   DATA[1296,24] := 2.0;
   DATA[1296,25] := 2.0;
   DATA[1296,26] := 7.87798;
   DATA[1296,27] := 143.0403;
   DATA[1296,28] := 263.0095;
   DATA[1296,29] := 11.88157;
   DATA[1296,30] := 1.726993;
   DATA[1296,31] := 1.274753;
   DATA[1296,32] := 0.7348846;
   DATA[1296,33] := 0.3082983;
   DATA[1296,34] := 2.0;
   DATA[1296,35] := 250.4646;
   DATA[1296,36] := 1.730048;
   DATA[1296,37] := 189.2624;
   DATA[1296,38] := 0.000128152;
   DATA[1296,39] := 1.0;
   DATA[1297,0] := 2.532428;
   DATA[1297,1] := 799.8927;
   DATA[1297,2] := 2.0;
   DATA[1297,3] := 1.0;
   DATA[1297,4] := 262.5609;
   DATA[1297,5] := 8.464369;
   DATA[1297,6] := 317.6878;
   DATA[1297,8] := 1.0;
   DATA[1297,9] := 1.0;
   DATA[1297,10] := 1.0;
   DATA[1297,11] := 1.997567;
   DATA[1297,12] := 0.000256221;
   DATA[1297,13] := 1010.879;
   DATA[1297,14] := 1.0;
   DATA[1297,15] := 1.0;
   DATA[1297,16] := 1.0;
   DATA[1297,17] := 1.0;
   DATA[1297,18] := 1.0;
   DATA[1297,19] := 1.0;
   DATA[1297,20] := 148.808;
   DATA[1297,21] := 153.8836;
   DATA[1297,22] := 1.716208;
   DATA[1297,23] := 809.6001;
   DATA[1297,24] := 2.0;
   DATA[1297,25] := 2.0;
   DATA[1297,26] := 7.87798;
   DATA[1297,27] := 143.0403;
   DATA[1297,28] := 263.0095;
   DATA[1297,29] := 12.07383;
   DATA[1297,30] := 1.726993;
   DATA[1297,31] := 1.277699;
   DATA[1297,32] := 0.7348846;
   DATA[1297,33] := 0.3082983;
   DATA[1297,34] := 2.0;
   DATA[1297,35] := 250.5447;
   DATA[1297,36] := 1.730048;
   DATA[1297,37] := 189.2624;
   DATA[1297,38] := 0.000128152;
   DATA[1297,39] := 1.0;
   DATA[1298,0] := 2.537873;
   DATA[1298,1] := 800.6385;
   DATA[1298,2] := 2.0;
   DATA[1298,3] := 1.0;
   DATA[1298,4] := 262.5609;
   DATA[1298,5] := 8.464369;
   DATA[1298,6] := 317.6878;
   DATA[1298,8] := 1.0;
   DATA[1298,9] := 1.0;
   DATA[1298,10] := 1.0;
   DATA[1298,11] := 1.997567;
   DATA[1298,12] := 0.000256221;
   DATA[1298,13] := 1010.879;
   DATA[1298,14] := 1.0;
   DATA[1298,15] := 1.0;
   DATA[1298,16] := 1.0;
   DATA[1298,17] := 1.0;
   DATA[1298,18] := 1.0;
   DATA[1298,19] := 1.0;
   DATA[1298,20] := 148.808;
   DATA[1298,21] := 153.8836;
   DATA[1298,22] := 1.716208;
   DATA[1298,23] := 809.1771;
   DATA[1298,24] := 2.0;
   DATA[1298,25] := 2.0;
   DATA[1298,26] := 7.87798;
   DATA[1298,27] := 143.0403;
   DATA[1298,28] := 263.0095;
   DATA[1298,29] := 12.07383;
   DATA[1298,30] := 1.726993;
   DATA[1298,31] := 1.274881;
   DATA[1298,32] := 0.7353967;
   DATA[1298,33] := 0.3082983;
   DATA[1298,34] := 2.0;
   DATA[1298,35] := 250.5447;
   DATA[1298,36] := 1.681991;
   DATA[1298,37] := 189.2624;
   DATA[1298,38] := 0.000128152;
   DATA[1298,39] := 1.0;
   DATA[1299,0] := 2.539474;
   DATA[1299,1] := 801.188;
   DATA[1299,3] := 1.0;
   DATA[1299,4] := 262.5609;
   DATA[1299,5] := 8.464369;
   DATA[1299,6] := 317.6878;
   DATA[1299,8] := 1.0;
   DATA[1299,9] := 1.0;
   DATA[1299,10] := 1.0;
   DATA[1299,11] := 1.997567;
   DATA[1299,12] := 0.000256221;
   DATA[1299,13] := 1010.758;
   DATA[1299,14] := 1.0;
   DATA[1299,15] := 1.0;
   DATA[1299,16] := 1.0;
   DATA[1299,17] := 1.0;
   DATA[1299,18] := 1.0;
   DATA[1299,19] := 1.0;
   DATA[1299,20] := 148.808;
   DATA[1299,21] := 153.8836;
   DATA[1299,22] := 1.717746;
   DATA[1299,23] := 809.1387;
   DATA[1299,24] := 2.0;
   DATA[1299,25] := 2.0;
   DATA[1299,26] := 7.87798;
   DATA[1299,27] := 143.0403;
   DATA[1299,28] := 263.0095;
   DATA[1299,29] := 12.07383;
   DATA[1299,30] := 1.726993;
   DATA[1299,31] := 1.291149;
   DATA[1299,32] := 0.7353967;
   DATA[1299,33] := 0.3082983;
   DATA[1299,34] := 2.0;
   DATA[1299,35] := 250.3525;
   DATA[1299,36] := 1.681991;
   DATA[1299,37] := 189.2624;
   DATA[1299,38] := 0.000128152;
   DATA[1299,39] := 1.0;
   DATA[1300,0] := 2.544278;
   DATA[1300,1] := 801.8161;
   DATA[1300,3] := 1.0;
   DATA[1300,4] := 262.5609;
   DATA[1300,5] := 8.464369;
   DATA[1300,6] := 317.6878;
   DATA[1300,8] := 1.0;
   DATA[1300,9] := 1.0;
   DATA[1300,10] := 1.0;
   DATA[1300,11] := 2.010372;
   DATA[1300,12] := 0.000256221;
   DATA[1300,13] := 1010.558;
   DATA[1300,14] := 1.0;
   DATA[1300,15] := 1.0;
   DATA[1300,16] := 1.0;
   DATA[1300,17] := 1.0;
   DATA[1300,18] := 1.0;
   DATA[1300,19] := 1.0;
   DATA[1300,20] := 148.808;
   DATA[1300,21] := 153.6785;
   DATA[1300,22] := 1.717746;
   DATA[1300,23] := 808.5619;
   DATA[1300,24] := 2.0;
   DATA[1300,25] := 2.0;
   DATA[1300,26] := 7.87798;
   DATA[1300,27] := 143.0403;
   DATA[1300,28] := 263.0095;
   DATA[1300,29] := 12.07383;
   DATA[1300,30] := 1.726993;
   DATA[1300,31] := 1.289996;
   DATA[1300,32] := 0.7353967;
   DATA[1300,33] := 0.3082983;
   DATA[1300,34] := 2.0;
   DATA[1300,35] := 250.3525;
   DATA[1300,36] := 1.681991;
   DATA[1300,37] := 189.2624;
   DATA[1300,38] := 0.000128152;
   DATA[1300,39] := 1.0;
   DATA[1301,0] := 2.54652;
   DATA[1301,1] := 802.5619;
   DATA[1301,3] := 1.0;
   DATA[1301,4] := 262.5609;
   DATA[1301,5] := 8.464369;
   DATA[1301,6] := 317.6878;
   DATA[1301,8] := 1.0;
   DATA[1301,9] := 1.0;
   DATA[1301,10] := 1.0;
   DATA[1301,11] := 2.010372;
   DATA[1301,12] := 0.000256221;
   DATA[1301,13] := 1010.678;
   DATA[1301,14] := 1.0;
   DATA[1301,15] := 1.0;
   DATA[1301,16] := 1.0;
   DATA[1301,17] := 1.0;
   DATA[1301,18] := 1.0;
   DATA[1301,19] := 1.0;
   DATA[1301,20] := 148.808;
   DATA[1301,21] := 153.6785;
   DATA[1301,22] := 1.717746;
   DATA[1301,23] := 808.1774;
   DATA[1301,24] := 2.0;
   DATA[1301,25] := 2.0;
   DATA[1301,26] := 7.87798;
   DATA[1301,27] := 143.0403;
   DATA[1301,28] := 263.0095;
   DATA[1301,29] := 12.07383;
   DATA[1301,30] := 1.726352;
   DATA[1301,31] := 1.28167;
   DATA[1301,32] := 0.7353967;
   DATA[1301,33] := 0.3082983;
   DATA[1301,34] := 2.0;
   DATA[1301,35] := 250.3525;
   DATA[1301,36] := 1.681991;
   DATA[1301,37] := 189.2624;
   DATA[1301,38] := 0.000128152;
   DATA[1301,39] := 1.0;
   DATA[1302,0] := 2.548762;
   DATA[1302,1] := 802.9544;
   DATA[1302,3] := 1.0;
   DATA[1302,4] := 262.5609;
   DATA[1302,5] := 8.464369;
   DATA[1302,6] := 317.6878;
   DATA[1302,8] := 1.0;
   DATA[1302,9] := 1.0;
   DATA[1302,10] := 1.0;
   DATA[1302,11] := 2.010372;
   DATA[1302,12] := 0.000256221;
   DATA[1302,13] := 1010.558;
   DATA[1302,14] := 1.0;
   DATA[1302,15] := 1.0;
   DATA[1302,16] := 1.0;
   DATA[1302,17] := 1.0;
   DATA[1302,18] := 1.0;
   DATA[1302,19] := 1.0;
   DATA[1302,20] := 148.808;
   DATA[1302,21] := 153.6785;
   DATA[1302,22] := 1.717746;
   DATA[1302,23] := 807.8313;
   DATA[1302,24] := 2.0;
   DATA[1302,25] := 2.0;
   DATA[1302,26] := 7.87798;
   DATA[1302,27] := 143.0403;
   DATA[1302,28] := 263.0095;
   DATA[1302,29] := 12.07383;
   DATA[1302,30] := 1.724686;
   DATA[1302,31] := 1.28167;
   DATA[1302,32] := 0.7353967;
   DATA[1302,33] := 0.3082983;
   DATA[1302,34] := 2.0;
   DATA[1302,35] := 250.3525;
   DATA[1302,36] := 1.681991;
   DATA[1302,37] := 189.2624;
   DATA[1302,38] := 0.000128152;
   DATA[1302,39] := 1.0;
   DATA[1303,0] := 2.548762;
   DATA[1303,1] := 803.9357;
   DATA[1303,3] := 1.0;
   DATA[1303,4] := 262.5609;
   DATA[1303,5] := 8.464369;
   DATA[1303,6] := 317.6878;
   DATA[1303,8] := 1.0;
   DATA[1303,9] := 1.0;
   DATA[1303,10] := 1.0;
   DATA[1303,11] := 2.010372;
   DATA[1303,12] := 0.000256221;
   DATA[1303,13] := 1010.678;
   DATA[1303,14] := 1.0;
   DATA[1303,15] := 1.0;
   DATA[1303,16] := 1.0;
   DATA[1303,17] := 1.0;
   DATA[1303,18] := 1.0;
   DATA[1303,19] := 1.0;
   DATA[1303,20] := 148.808;
   DATA[1303,21] := 153.6785;
   DATA[1303,22] := 1.717746;
   DATA[1303,23] := 807.4468;
   DATA[1303,24] := 2.0;
   DATA[1303,25] := 2.0;
   DATA[1303,26] := 7.87798;
   DATA[1303,27] := 143.0403;
   DATA[1303,28] := 263.0095;
   DATA[1303,29] := 12.07383;
   DATA[1303,30] := 1.724686;
   DATA[1303,31] := 1.274497;
   DATA[1303,32] := 0.7353967;
   DATA[1303,33] := 0.3082983;
   DATA[1303,34] := 2.0;
   DATA[1303,35] := 250.3525;
   DATA[1303,36] := 1.681991;
   DATA[1303,37] := 189.2624;
   DATA[1303,38] := 0.000128152;
   DATA[1303,39] := 1.0;
   DATA[1304,0] := 2.537873;
   DATA[1304,1] := 804.4068;
   DATA[1304,3] := 1.0;
   DATA[1304,4] := 262.5609;
   DATA[1304,5] := 8.464369;
   DATA[1304,6] := 317.6878;
   DATA[1304,8] := 1.0;
   DATA[1304,9] := 1.0;
   DATA[1304,10] := 1.0;
   DATA[1304,11] := 2.010372;
   DATA[1304,12] := 0.000256221;
   DATA[1304,13] := 1010.959;
   DATA[1304,14] := 1.0;
   DATA[1304,15] := 1.0;
   DATA[1304,16] := 1.0;
   DATA[1304,17] := 1.0;
   DATA[1304,18] := 1.0;
   DATA[1304,19] := 1.0;
   DATA[1304,20] := 148.808;
   DATA[1304,21] := 153.6785;
   DATA[1304,22] := 1.717746;
   DATA[1304,23] := 807.4853;
   DATA[1304,24] := 2.0;
   DATA[1304,25] := 2.0;
   DATA[1304,26] := 7.87798;
   DATA[1304,27] := 143.0403;
   DATA[1304,28] := 263.0095;
   DATA[1304,29] := 12.07383;
   DATA[1304,30] := 1.724686;
   DATA[1304,31] := 1.277315;
   DATA[1304,32] := 0.7353967;
   DATA[1304,33] := 0.3082983;
   DATA[1304,34] := 2.0;
   DATA[1304,35] := 250.3525;
   DATA[1304,36] := 1.681991;
   DATA[1304,37] := 189.2624;
   DATA[1304,38] := 0.000128152;
   DATA[1304,39] := 1.0;
   DATA[1305,0] := 2.515133;
   DATA[1305,1] := 804.9171;
   DATA[1305,3] := 1.0;
   DATA[1305,4] := 262.5609;
   DATA[1305,5] := 8.464369;
   DATA[1305,6] := 317.6878;
   DATA[1305,8] := 1.0;
   DATA[1305,9] := 1.0;
   DATA[1305,10] := 1.0;
   DATA[1305,11] := 2.010372;
   DATA[1305,12] := 0.000256221;
   DATA[1305,13] := 1010.919;
   DATA[1305,14] := 1.0;
   DATA[1305,15] := 1.0;
   DATA[1305,16] := 1.0;
   DATA[1305,17] := 1.0;
   DATA[1305,18] := 1.0;
   DATA[1305,19] := 1.0;
   DATA[1305,20] := 148.808;
   DATA[1305,21] := 153.6785;
   DATA[1305,22] := 1.717746;
   DATA[1305,23] := 806.9085;
   DATA[1305,24] := 2.0;
   DATA[1305,25] := 2.0;
   DATA[1305,26] := 7.87798;
   DATA[1305,27] := 143.0403;
   DATA[1305,28] := 263.0095;
   DATA[1305,29] := 12.07383;
   DATA[1305,30] := 1.724686;
   DATA[1305,31] := 1.291789;
   DATA[1305,32] := 0.7353967;
   DATA[1305,33] := 0.3082983;
   DATA[1305,34] := 2.0;
   DATA[1305,35] := 250.3525;
   DATA[1305,36] := 1.681991;
   DATA[1305,37] := 189.2624;
   DATA[1305,38] := 0.000128152;
   DATA[1305,39] := 1.0;
   DATA[1306,0] := 2.464209;
   DATA[1306,1] := 805.5451;
   DATA[1306,3] := 1.0;
   DATA[1306,4] := 262.5609;
   DATA[1306,5] := 8.464369;
   DATA[1306,6] := 317.6878;
   DATA[1306,8] := 1.0;
   DATA[1306,9] := 1.0;
   DATA[1306,10] := 1.0;
   DATA[1306,11] := 2.010372;
   DATA[1306,12] := 0.000256221;
   DATA[1306,13] := 1011.119;
   DATA[1306,14] := 1.0;
   DATA[1306,15] := 1.0;
   DATA[1306,16] := 1.0;
   DATA[1306,17] := 1.0;
   DATA[1306,18] := 1.0;
   DATA[1306,19] := 1.0;
   DATA[1306,20] := 148.808;
   DATA[1306,21] := 153.6785;
   DATA[1306,22] := 1.717746;
   DATA[1306,23] := 806.2933;
   DATA[1306,24] := 2.0;
   DATA[1306,25] := 2.0;
   DATA[1306,26] := 7.87798;
   DATA[1306,27] := 143.0403;
   DATA[1306,28] := 263.0095;
   DATA[1306,29] := 12.07383;
   DATA[1306,30] := 1.724686;
   DATA[1306,31] := 1.301652;
   DATA[1306,32] := 0.7353967;
   DATA[1306,33] := 0.3082983;
   DATA[1306,34] := 2.0;
   DATA[1306,35] := 250.3525;
   DATA[1306,36] := 1.746067;
   DATA[1306,37] := 189.2624;
   DATA[1306,38] := 0.000128152;
   DATA[1306,39] := 1.0;
   DATA[1307,0] := 2.393428;
   DATA[1307,1] := 805.9769;
   DATA[1307,2] := 1.0;
   DATA[1307,3] := 1.0;
   DATA[1307,4] := 262.5609;
   DATA[1307,5] := 8.464369;
   DATA[1307,6] := 317.6878;
   DATA[1307,8] := 1.0;
   DATA[1307,9] := 1.0;
   DATA[1307,10] := 1.0;
   DATA[1307,11] := 2.010372;
   DATA[1307,12] := 0.000256221;
   DATA[1307,13] := 1010.758;
   DATA[1307,14] := 1.0;
   DATA[1307,15] := 1.0;
   DATA[1307,16] := 1.0;
   DATA[1307,17] := 1.0;
   DATA[1307,18] := 1.0;
   DATA[1307,19] := 1.0;
   DATA[1307,20] := 148.808;
   DATA[1307,21] := 153.8067;
   DATA[1307,22] := 1.717746;
   DATA[1307,23] := 805.7934;
   DATA[1307,24] := 2.0;
   DATA[1307,25] := 2.0;
   DATA[1307,26] := 7.87798;
   DATA[1307,27] := 143.0403;
   DATA[1307,28] := 263.0095;
   DATA[1307,29] := 12.07383;
   DATA[1307,30] := 1.724686;
   DATA[1307,31] := 1.302677;
   DATA[1307,32] := 0.7353967;
   DATA[1307,33] := 0.3082983;
   DATA[1307,34] := 2.0;
   DATA[1307,35] := 250.3525;
   DATA[1307,36] := 1.746067;
   DATA[1307,37] := 189.2624;
   DATA[1307,38] := 0.000128152;
   DATA[1307,39] := 1.0;
   DATA[1308,0] := 2.276206;
   DATA[1308,1] := 806.2516;
   DATA[1308,2] := 1.0;
   DATA[1308,3] := 1.0;
   DATA[1308,4] := 262.5609;
   DATA[1308,5] := 8.464369;
   DATA[1308,6] := 317.6878;
   DATA[1308,8] := 1.0;
   DATA[1308,9] := 1.0;
   DATA[1308,10] := 1.0;
   DATA[1308,11] := 2.010372;
   DATA[1308,12] := 0.000256221;
   DATA[1308,13] := 1011.079;
   DATA[1308,14] := 1.0;
   DATA[1308,15] := 1.0;
   DATA[1308,16] := 1.0;
   DATA[1308,17] := 1.0;
   DATA[1308,18] := 1.0;
   DATA[1308,19] := 1.0;
   DATA[1308,20] := 148.808;
   DATA[1308,21] := 153.8067;
   DATA[1308,22] := 1.717746;
   DATA[1308,23] := 805.7934;
   DATA[1308,24] := 2.0;
   DATA[1308,25] := 2.0;
   DATA[1308,26] := 7.87798;
   DATA[1308,27] := 143.0403;
   DATA[1308,28] := 263.0095;
   DATA[1308,29] := 12.07383;
   DATA[1308,30] := 1.724686;
   DATA[1308,31] := 1.310747;
   DATA[1308,32] := 0.7353967;
   DATA[1308,33] := 0.3082983;
   DATA[1308,34] := 2.0;
   DATA[1308,35] := 250.3525;
   DATA[1308,36] := 1.746067;
   DATA[1308,37] := 189.2624;
   DATA[1308,38] := 0.000128152;
   DATA[1308,39] := 1.0;
   DATA[1309,0] := 2.053935;
   DATA[1309,1] := 806.6442;
   DATA[1309,2] := 1.0;
   DATA[1309,3] := 1.0;
   DATA[1309,4] := 262.5609;
   DATA[1309,5] := 8.464369;
   DATA[1309,6] := 317.6878;
   DATA[1309,8] := 1.0;
   DATA[1309,9] := 1.0;
   DATA[1309,10] := 1.0;
   DATA[1309,11] := 2.010372;
   DATA[1309,12] := 0.000256221;
   DATA[1309,13] := 1011.159;
   DATA[1309,14] := 1.0;
   DATA[1309,15] := 1.0;
   DATA[1309,16] := 1.0;
   DATA[1309,17] := 1.0;
   DATA[1309,18] := 1.0;
   DATA[1309,19] := 1.0;
   DATA[1309,20] := 148.808;
   DATA[1309,21] := 153.8067;
   DATA[1309,22] := 1.717746;
   DATA[1309,23] := 805.1397;
   DATA[1309,24] := 2.0;
   DATA[1309,25] := 2.0;
   DATA[1309,26] := 7.87798;
   DATA[1309,27] := 143.0403;
   DATA[1309,28] := 263.0095;
   DATA[1309,29] := 12.07383;
   DATA[1309,30] := 1.724045;
   DATA[1309,31] := 1.312028;
   DATA[1309,32] := 0.7353967;
   DATA[1309,33] := 0.3082983;
   DATA[1309,34] := 2.0;
   DATA[1309,35] := 250.3525;
   DATA[1309,36] := 1.746067;
   DATA[1309,37] := 189.2624;
   DATA[1309,38] := 0.000128152;
   DATA[1309,39] := 1.0;
   DATA[1310,0] := 1.653268;
   DATA[1310,1] := 807.3115;
   DATA[1310,2] := 1.0;
   DATA[1310,3] := 1.0;
   DATA[1310,4] := 262.5609;
   DATA[1310,5] := 8.464369;
   DATA[1310,6] := 317.6878;
   DATA[1310,8] := 1.0;
   DATA[1310,9] := 1.0;
   DATA[1310,10] := 1.0;
   DATA[1310,11] := 2.010372;
   DATA[1310,12] := 0.000256221;
   DATA[1310,13] := 1010.678;
   DATA[1310,14] := 1.0;
   DATA[1310,15] := 1.0;
   DATA[1310,16] := 1.0;
   DATA[1310,17] := 1.0;
   DATA[1310,18] := 1.0;
   DATA[1310,19] := 1.0;
   DATA[1310,20] := 148.808;
   DATA[1310,21] := 153.8067;
   DATA[1310,22] := 1.717746;
   DATA[1310,23] := 804.6398;
   DATA[1310,24] := 2.0;
   DATA[1310,25] := 2.0;
   DATA[1310,26] := 7.87798;
   DATA[1310,27] := 143.0403;
   DATA[1310,28] := 263.0095;
   DATA[1310,29] := 12.07383;
   DATA[1310,30] := 1.724045;
   DATA[1310,31] := 1.305367;
   DATA[1310,32] := 0.7353967;
   DATA[1310,33] := 0.3082983;
   DATA[1310,34] := 2.0;
   DATA[1310,35] := 250.3525;
   DATA[1310,36] := 1.746067;
   DATA[1310,37] := 189.2624;
   DATA[1310,38] := 0.000128152;
   DATA[1310,39] := 1.0;
   DATA[1311,0] := 1.308651;
   DATA[1311,1] := 807.7432;
   DATA[1311,2] := 1.0;
   DATA[1311,3] := 1.0;
   DATA[1311,4] := 262.5609;
   DATA[1311,5] := 8.464369;
   DATA[1311,6] := 317.6878;
   DATA[1311,8] := 1.0;
   DATA[1311,9] := 1.0;
   DATA[1311,10] := 1.0;
   DATA[1311,11] := 2.010372;
   DATA[1311,12] := 0.000256221;
   DATA[1311,13] := 1010.879;
   DATA[1311,14] := 1.0;
   DATA[1311,15] := 1.0;
   DATA[1311,16] := 1.0;
   DATA[1311,17] := 1.0;
   DATA[1311,18] := 1.0;
   DATA[1311,19] := 1.0;
   DATA[1311,20] := 148.808;
   DATA[1311,21] := 153.8067;
   DATA[1311,22] := 1.717746;
   DATA[1311,23] := 804.0246;
   DATA[1311,24] := 2.0;
   DATA[1311,25] := 2.0;
   DATA[1311,26] := 7.87798;
   DATA[1311,27] := 143.0403;
   DATA[1311,28] := 263.0095;
   DATA[1311,29] := 12.07383;
   DATA[1311,30] := 1.724045;
   DATA[1311,31] := 1.302805;
   DATA[1311,32] := 0.7353967;
   DATA[1311,33] := 0.3084265;
   DATA[1311,34] := 2.0;
   DATA[1311,35] := 250.3525;
   DATA[1311,36] := 1.746067;
   DATA[1311,37] := 189.2624;
   DATA[1311,38] := 0.000128152;
   DATA[1311,39] := 1.0;
   DATA[1312,0] := 0.9060628;
   DATA[1312,1] := 808.2928;
   DATA[1312,2] := 1.0;
   DATA[1312,3] := 1.0;
   DATA[1312,4] := 262.5609;
   DATA[1312,5] := 8.464369;
   DATA[1312,6] := 317.6878;
   DATA[1312,8] := 1.0;
   DATA[1312,9] := 1.0;
   DATA[1312,10] := 1.0;
   DATA[1312,11] := 2.010372;
   DATA[1312,13] := 1010.638;
   DATA[1312,14] := 1.0;
   DATA[1312,15] := 1.0;
   DATA[1312,16] := 1.0;
   DATA[1312,17] := 1.0;
   DATA[1312,18] := 1.0;
   DATA[1312,19] := 1.0;
   DATA[1312,20] := 148.808;
   DATA[1312,21] := 153.8067;
   DATA[1312,22] := 1.717489;
   DATA[1312,23] := 804.0246;
   DATA[1312,24] := 2.0;
   DATA[1312,25] := 2.0;
   DATA[1312,26] := 7.87798;
   DATA[1312,27] := 143.0403;
   DATA[1312,28] := 263.0095;
   DATA[1312,29] := 12.07383;
   DATA[1312,30] := 1.722123;
   DATA[1312,31] := 1.282567;
   DATA[1312,32] := 0.7353967;
   DATA[1312,33] := 0.3084265;
   DATA[1312,34] := 2.0;
   DATA[1312,35] := 250.3525;
   DATA[1312,36] := 1.746067;
   DATA[1312,37] := 189.1662;
   DATA[1312,38] := 0.000128152;
   DATA[1312,39] := 1.0;
   DATA[1313,0] := 0.5736156;
   DATA[1313,1] := 808.7245;
   DATA[1313,2] := 1.0;
   DATA[1313,3] := 1.0;
   DATA[1313,4] := 262.5609;
   DATA[1313,5] := 8.464369;
   DATA[1313,6] := 317.6878;
   DATA[1313,8] := 1.0;
   DATA[1313,9] := 1.0;
   DATA[1313,10] := 1.0;
   DATA[1313,11] := 2.010372;
   DATA[1313,13] := 1011.079;
   DATA[1313,14] := 1.0;
   DATA[1313,15] := 1.0;
   DATA[1313,16] := 1.0;
   DATA[1313,17] := 1.0;
   DATA[1313,18] := 1.0;
   DATA[1313,19] := 1.0;
   DATA[1313,20] := 148.808;
   DATA[1313,21] := 153.8067;
   DATA[1313,22] := 1.715439;
   DATA[1313,23] := 803.1786;
   DATA[1313,24] := 2.0;
   DATA[1313,25] := 2.0;
   DATA[1313,26] := 7.87798;
   DATA[1313,27] := 143.0403;
   DATA[1313,28] := 263.0095;
   DATA[1313,29] := 12.07383;
   DATA[1313,30] := 1.722123;
   DATA[1313,31] := 1.261688;
   DATA[1313,32] := 0.7353967;
   DATA[1313,33] := 0.3084265;
   DATA[1313,34] := 2.0;
   DATA[1313,35] := 250.0961;
   DATA[1313,36] := 1.746067;
   DATA[1313,37] := 188.9259;
   DATA[1313,38] := 0.000128152;
   DATA[1313,39] := 1.0;
   DATA[1314,0] := 0.3468597;
   DATA[1314,1] := 809.5096;
   DATA[1314,2] := 1.0;
   DATA[1314,3] := 1.0;
   DATA[1314,4] := 262.5609;
   DATA[1314,5] := 8.464369;
   DATA[1314,6] := 317.7903;
   DATA[1314,8] := 1.0;
   DATA[1314,9] := 1.0;
   DATA[1314,10] := 1.0;
   DATA[1314,11] := 2.010372;
   DATA[1314,13] := 1010.839;
   DATA[1314,14] := 1.0;
   DATA[1314,15] := 1.0;
   DATA[1314,16] := 1.0;
   DATA[1314,17] := 1.0;
   DATA[1314,18] := 1.0;
   DATA[1314,19] := 1.0;
   DATA[1314,20] := 148.808;
   DATA[1314,21] := 153.8067;
   DATA[1314,22] := 1.711979;
   DATA[1314,23] := 803.0248;
   DATA[1314,24] := 2.0;
   DATA[1314,25] := 2.0;
   DATA[1314,26] := 7.87798;
   DATA[1314,27] := 143.0403;
   DATA[1314,28] := 263.0095;
   DATA[1314,29] := 12.07383;
   DATA[1314,30] := 1.722123;
   DATA[1314,31] := 1.254643;
   DATA[1314,32] := 0.7353967;
   DATA[1314,33] := 0.3084265;
   DATA[1314,34] := 2.0;
   DATA[1314,35] := 249.9359;
   DATA[1314,36] := 1.778105;
   DATA[1314,37] := 188.8138;
   DATA[1314,38] := 0.000128152;
   DATA[1314,39] := 1.0;
   DATA[1315,0] := 0.1896038;
   DATA[1315,1] := 810.2162;
   DATA[1315,2] := 1.0;
   DATA[1315,3] := 1.0;
   DATA[1315,4] := 262.5609;
   DATA[1315,5] := 8.464369;
   DATA[1315,6] := 317.7903;
   DATA[1315,8] := 1.0;
   DATA[1315,9] := 1.0;
   DATA[1315,10] := 1.0;
   DATA[1315,11] := 2.010372;
   DATA[1315,13] := 1011.119;
   DATA[1315,14] := 1.0;
   DATA[1315,15] := 1.0;
   DATA[1315,16] := 1.0;
   DATA[1315,17] := 1.0;
   DATA[1315,18] := 1.0;
   DATA[1315,19] := 1.0;
   DATA[1315,20] := 148.808;
   DATA[1315,21] := 153.8067;
   DATA[1315,22] := 1.711338;
   DATA[1315,23] := 802.6788;
   DATA[1315,24] := 2.0;
   DATA[1315,25] := 2.0;
   DATA[1315,26] := 7.87798;
   DATA[1315,27] := 143.0403;
   DATA[1315,28] := 263.0095;
   DATA[1315,29] := 12.07383;
   DATA[1315,30] := 1.722123;
   DATA[1315,31] := 1.261048;
   DATA[1315,32] := 0.7353967;
   DATA[1315,33] := 0.3084265;
   DATA[1315,34] := 2.0;
   DATA[1315,35] := 249.9359;
   DATA[1315,36] := 1.778105;
   DATA[1315,37] := 188.8138;
   DATA[1315,38] := 0.000128152;
   DATA[1315,39] := 1.0;
   DATA[1316,0] := 0.09191941;
   DATA[1316,1] := 810.6087;
   DATA[1316,2] := 1.0;
   DATA[1316,3] := 1.0;
   DATA[1316,4] := 262.5609;
   DATA[1316,5] := 8.464369;
   DATA[1316,6] := 317.7903;
   DATA[1316,8] := 1.0;
   DATA[1316,9] := 1.0;
   DATA[1316,10] := 1.0;
   DATA[1316,11] := 2.010372;
   DATA[1316,13] := 1010.839;
   DATA[1316,14] := 1.0;
   DATA[1316,15] := 1.0;
   DATA[1316,16] := 1.0;
   DATA[1316,17] := 1.0;
   DATA[1316,18] := 1.0;
   DATA[1316,19] := 1.0;
   DATA[1316,20] := 148.808;
   DATA[1316,21] := 153.8067;
   DATA[1316,22] := 1.710698;
   DATA[1316,23] := 801.9098;
   DATA[1316,24] := 2.0;
   DATA[1316,25] := 2.0;
   DATA[1316,26] := 7.87798;
   DATA[1316,27] := 143.0403;
   DATA[1316,28] := 263.0095;
   DATA[1316,29] := 12.07383;
   DATA[1316,30] := 1.722123;
   DATA[1316,31] := 1.270655;
   DATA[1316,32] := 0.7353967;
   DATA[1316,33] := 0.3104122;
   DATA[1316,34] := 2.0;
   DATA[1316,35] := 249.9359;
   DATA[1316,36] := 1.778105;
   DATA[1316,37] := 188.8138;
   DATA[1316,38] := 0.000128152;
   DATA[1316,39] := 1.0;
   DATA[1317,0] := 0.0425968;
   DATA[1317,1] := 810.805;
   DATA[1317,2] := 1.0;
   DATA[1317,3] := 1.0;
   DATA[1317,4] := 262.5609;
   DATA[1317,5] := 8.464369;
   DATA[1317,6] := 317.7903;
   DATA[1317,8] := 1.0;
   DATA[1317,9] := 1.0;
   DATA[1317,10] := 1.0;
   DATA[1317,11] := 2.010372;
   DATA[1317,13] := 1010.678;
   DATA[1317,14] := 1.0;
   DATA[1317,15] := 1.0;
   DATA[1317,16] := 1.0;
   DATA[1317,17] := 1.0;
   DATA[1317,18] := 1.0;
   DATA[1317,19] := 1.0;
   DATA[1317,20] := 148.808;
   DATA[1317,21] := 153.8067;
   DATA[1317,22] := 1.710698;
   DATA[1317,23] := 801.1407;
   DATA[1317,24] := 2.0;
   DATA[1317,25] := 2.0;
   DATA[1317,26] := 7.87798;
   DATA[1317,27] := 143.0403;
   DATA[1317,28] := 263.0095;
   DATA[1317,29] := 12.07383;
   DATA[1317,30] := 1.722123;
   DATA[1317,31] := 1.27232;
   DATA[1317,32] := 0.7353967;
   DATA[1317,33] := 0.3106684;
   DATA[1317,34] := 2.0;
   DATA[1317,35] := 249.9359;
   DATA[1317,36] := 1.778105;
   DATA[1317,37] := 188.8138;
   DATA[1317,38] := 0.000128152;
   DATA[1317,39] := 1.0;
   DATA[1318,0] := 0.001281107;
   DATA[1318,1] := 811.0797;
   DATA[1318,2] := 1.0;
   DATA[1318,3] := 1.0;
   DATA[1318,4] := 262.5609;
   DATA[1318,5] := 8.464369;
   DATA[1318,6] := 317.7903;
   DATA[1318,8] := 1.0;
   DATA[1318,9] := 1.0;
   DATA[1318,10] := 1.0;
   DATA[1318,11] := 2.010372;
   DATA[1318,13] := 1011.039;
   DATA[1318,14] := 1.0;
   DATA[1318,15] := 1.0;
   DATA[1318,16] := 1.0;
   DATA[1318,17] := 1.0;
   DATA[1318,18] := 1.0;
   DATA[1318,19] := 1.0;
   DATA[1318,20] := 148.808;
   DATA[1318,21] := 153.8067;
   DATA[1318,22] := 1.710698;
   DATA[1318,23] := 800.8716;
   DATA[1318,24] := 2.0;
   DATA[1318,25] := 2.0;
   DATA[1318,26] := 7.87798;
   DATA[1318,27] := 143.0403;
   DATA[1318,28] := 263.0095;
   DATA[1318,29] := 12.07383;
   DATA[1318,30] := 1.722123;
   DATA[1318,31] := 1.27232;
   DATA[1318,32] := 0.7353967;
   DATA[1318,33] := 0.3106684;
   DATA[1318,34] := 2.0;
   DATA[1318,35] := 249.8718;
   DATA[1318,36] := 1.778105;
   DATA[1318,37] := 188.8138;
   DATA[1318,38] := 0.000128152;
   DATA[1318,39] := 1.0;
   DATA[1319,0] := 0.000640553;
   DATA[1319,1] := 811.6685;
   DATA[1319,2] := 1.0;
   DATA[1319,3] := 1.0;
   DATA[1319,4] := 262.5609;
   DATA[1319,5] := 8.464369;
   DATA[1319,6] := 317.7903;
   DATA[1319,8] := 1.0;
   DATA[1319,9] := 1.0;
   DATA[1319,10] := 1.0;
   DATA[1319,11] := 2.010372;
   DATA[1319,12] := 0.000384332;
   DATA[1319,13] := 1010.919;
   DATA[1319,14] := 1.0;
   DATA[1319,15] := 1.0;
   DATA[1319,16] := 1.0;
   DATA[1319,17] := 1.0;
   DATA[1319,18] := 1.0;
   DATA[1319,19] := 1.0;
   DATA[1319,20] := 148.808;
   DATA[1319,21] := 153.8067;
   DATA[1319,22] := 1.710698;
   DATA[1319,23] := 800.1794;
   DATA[1319,24] := 2.0;
   DATA[1319,25] := 2.0;
   DATA[1319,26] := 7.87798;
   DATA[1319,27] := 143.1684;
   DATA[1319,28] := 263.0095;
   DATA[1319,29] := 12.07383;
   DATA[1319,30] := 1.722123;
   DATA[1319,31] := 1.27232;
   DATA[1319,32] := 0.7353967;
   DATA[1319,33] := 0.3106684;
   DATA[1319,34] := 2.0;
   DATA[1319,35] := 249.8718;
   DATA[1319,36] := 1.617916;
   DATA[1319,37] := 188.6055;
   DATA[1319,38] := 0.000128152;
   DATA[1319,39] := 1.0;
   DATA[1320,1] := 812.2181;
   DATA[1320,2] := 1.0;
   DATA[1320,3] := 1.0;
   DATA[1320,4] := 262.5609;
   DATA[1320,5] := 8.464369;
   DATA[1320,6] := 318.0723;
   DATA[1320,8] := 1.0;
   DATA[1320,9] := 1.0;
   DATA[1320,10] := 1.0;
   DATA[1320,11] := 2.010372;
   DATA[1320,12] := 0.000384332;
   DATA[1320,13] := 1011.159;
   DATA[1320,14] := 1.0;
   DATA[1320,15] := 1.0;
   DATA[1320,16] := 1.0;
   DATA[1320,17] := 1.0;
   DATA[1320,18] := 1.0;
   DATA[1320,19] := 1.0;
   DATA[1320,20] := 148.808;
   DATA[1320,21] := 154.0118;
   DATA[1320,22] := 1.710698;
   DATA[1320,23] := 799.9872;
   DATA[1320,24] := 2.0;
   DATA[1320,25] := 2.0;
   DATA[1320,26] := 7.87798;
   DATA[1320,27] := 143.1684;
   DATA[1320,28] := 263.0095;
   DATA[1320,29] := 12.07383;
   DATA[1320,30] := 1.722123;
   DATA[1320,31] := 1.27232;
   DATA[1320,32] := 0.7353967;
   DATA[1320,33] := 0.3106684;
   DATA[1320,34] := 2.0;
   DATA[1320,35] := 249.8718;
   DATA[1320,36] := 1.617916;
   DATA[1320,37] := 188.6055;
   DATA[1320,38] := 0.000128152;
   DATA[1320,39] := 1.0;
   DATA[1321,1] := 812.3751;
   DATA[1321,2] := 1.0;
   DATA[1321,3] := 1.0;
   DATA[1321,4] := 262.5609;
   DATA[1321,5] := 8.464369;
   DATA[1321,6] := 318.0723;
   DATA[1321,8] := 1.0;
   DATA[1321,9] := 1.0;
   DATA[1321,10] := 1.0;
   DATA[1321,11] := 2.010372;
   DATA[1321,12] := 0.000384332;
   DATA[1321,13] := 1011.119;
   DATA[1321,14] := 1.0;
   DATA[1321,15] := 1.0;
   DATA[1321,16] := 1.0;
   DATA[1321,17] := 1.0;
   DATA[1321,18] := 1.0;
   DATA[1321,19] := 1.0;
   DATA[1321,20] := 148.808;
   DATA[1321,21] := 154.0118;
   DATA[1321,22] := 1.710698;
   DATA[1321,23] := 799.3719;
   DATA[1321,24] := 2.0;
   DATA[1321,25] := 2.0;
   DATA[1321,26] := 7.87798;
   DATA[1321,27] := 143.1684;
   DATA[1321,28] := 263.0095;
   DATA[1321,29] := 12.07383;
   DATA[1321,30] := 1.722123;
   DATA[1321,31] := 1.27232;
   DATA[1321,32] := 0.7353967;
   DATA[1321,33] := 0.3088108;
   DATA[1321,34] := 2.0;
   DATA[1321,35] := 249.7597;
   DATA[1321,36] := 1.617916;
   DATA[1321,37] := 188.6055;
   DATA[1321,38] := 0.000128152;
   DATA[1321,39] := 1.0;
   DATA[1322,1] := 812.8069;
   DATA[1322,2] := 1.0;
   DATA[1322,3] := 1.0;
   DATA[1322,4] := 262.5609;
   DATA[1322,5] := 8.464369;
   DATA[1322,6] := 318.0723;
   DATA[1322,8] := 1.0;
   DATA[1322,9] := 1.0;
   DATA[1322,10] := 1.0;
   DATA[1322,11] := 2.010372;
   DATA[1322,12] := 0.000384332;
   DATA[1322,13] := 1011.159;
   DATA[1322,14] := 1.0;
   DATA[1322,15] := 1.0;
   DATA[1322,16] := 1.0;
   DATA[1322,18] := 1.0;
   DATA[1322,19] := 1.0;
   DATA[1322,20] := 148.808;
   DATA[1322,21] := 154.0118;
   DATA[1322,22] := 1.713517;
   DATA[1322,23] := 799.6411;
   DATA[1322,24] := 2.0;
   DATA[1322,25] := 2.0;
   DATA[1322,26] := 7.87798;
   DATA[1322,27] := 143.1684;
   DATA[1322,28] := 263.0095;
   DATA[1322,29] := 12.07383;
   DATA[1322,30] := 1.723661;
   DATA[1322,31] := 1.268989;
   DATA[1322,32] := 0.7353967;
   DATA[1322,33] := 0.3086827;
   DATA[1322,34] := 2.0;
   DATA[1322,35] := 249.7597;
   DATA[1322,36] := 1.617916;
   DATA[1322,37] := 188.6856;
   DATA[1322,38] := 0.000128152;
   DATA[1322,39] := 1.0;
   DATA[1323,1] := 813.4349;
   DATA[1323,2] := 1.0;
   DATA[1323,3] := 1.0;
   DATA[1323,4] := 262.5609;
   DATA[1323,5] := 8.464369;
   DATA[1323,6] := 317.9185;
   DATA[1323,8] := 1.0;
   DATA[1323,9] := 1.0;
   DATA[1323,10] := 1.0;
   DATA[1323,11] := 2.010372;
   DATA[1323,12] := 0.000384332;
   DATA[1323,13] := 1011.039;
   DATA[1323,14] := 1.0;
   DATA[1323,15] := 1.0;
   DATA[1323,16] := 1.0;
   DATA[1323,18] := 1.0;
   DATA[1323,19] := 1.0;
   DATA[1323,20] := 148.808;
   DATA[1323,21] := 154.0118;
   DATA[1323,22] := 1.713517;
   DATA[1323,23] := 798.9874;
   DATA[1323,24] := 2.0;
   DATA[1323,25] := 2.0;
   DATA[1323,26] := 7.87798;
   DATA[1323,27] := 142.9633;
   DATA[1323,28] := 263.0095;
   DATA[1323,29] := 12.07383;
   DATA[1323,30] := 1.723789;
   DATA[1323,31] := 1.262329;
   DATA[1323,32] := 0.7360369;
   DATA[1323,33] := 0.3083624;
   DATA[1323,34] := 2.0;
   DATA[1323,35] := 249.7597;
   DATA[1323,36] := 1.617916;
   DATA[1323,37] := 188.6856;
   DATA[1323,38] := 0.000128152;
   DATA[1323,39] := 1.0;
   DATA[1324,1] := 813.3564;
   DATA[1324,2] := 1.0;
   DATA[1324,3] := 1.0;
   DATA[1324,4] := 262.5609;
   DATA[1324,5] := 8.464369;
   DATA[1324,6] := 317.9185;
   DATA[1324,8] := 1.0;
   DATA[1324,9] := 1.0;
   DATA[1324,10] := 1.0;
   DATA[1324,11] := 1.658237;
   DATA[1324,12] := 0.000384332;
   DATA[1324,13] := 1010.919;
   DATA[1324,14] := 1.0;
   DATA[1324,15] := 1.0;
   DATA[1324,16] := 1.0;
   DATA[1324,18] := 1.0;
   DATA[1324,19] := 1.0;
   DATA[1324,20] := 148.808;
   DATA[1324,21] := 154.0118;
   DATA[1324,22] := 1.713517;
   DATA[1324,23] := 798.8721;
   DATA[1324,24] := 2.0;
   DATA[1324,25] := 2.0;
   DATA[1324,26] := 7.87798;
   DATA[1324,27] := 142.9633;
   DATA[1324,28] := 263.0095;
   DATA[1324,29] := 12.07383;
   DATA[1324,30] := 1.723789;
   DATA[1324,31] := 1.267068;
   DATA[1324,32] := 0.736421;
   DATA[1324,33] := 0.3081703;
   DATA[1324,34] := 2.0;
   DATA[1324,35] := 249.7597;
   DATA[1324,36] := 1.617916;
   DATA[1324,37] := 188.6856;
   DATA[1324,38] := 0.000128152;
   DATA[1324,39] := 1.0;
   DATA[1325,1] := 813.5527;
   DATA[1325,2] := 1.0;
   DATA[1325,3] := 1.0;
   DATA[1325,4] := 262.5609;
   DATA[1325,5] := 8.464369;
   DATA[1325,6] := 317.9185;
   DATA[1325,8] := 1.0;
   DATA[1325,9] := 1.0;
   DATA[1325,10] := 1.0;
   DATA[1325,11] := 1.264486;
   DATA[1325,12] := 0.000384332;
   DATA[1325,13] := 1010.718;
   DATA[1325,14] := 1.0;
   DATA[1325,15] := 1.0;
   DATA[1325,16] := 1.0;
   DATA[1325,18] := 1.0;
   DATA[1325,19] := 1.0;
   DATA[1325,20] := 148.808;
   DATA[1325,21] := 154.0118;
   DATA[1325,22] := 1.713517;
   DATA[1325,23] := 798.6798;
   DATA[1325,24] := 2.0;
   DATA[1325,25] := 2.0;
   DATA[1325,26] := 7.87798;
   DATA[1325,27] := 142.9633;
   DATA[1325,28] := 263.0095;
   DATA[1325,29] := 12.07383;
   DATA[1325,30] := 1.723789;
   DATA[1325,31] := 1.266171;
   DATA[1325,32] := 0.736421;
   DATA[1325,33] := 0.3081703;
   DATA[1325,34] := 2.0;
   DATA[1325,35] := 249.7597;
   DATA[1325,36] := 1.617916;
   DATA[1325,37] := 188.6856;
   DATA[1325,38] := 0.000128152;
   DATA[1325,39] := 1.0;
   DATA[1326,1] := 813.7097;
   DATA[1326,2] := 1.0;
   DATA[1326,3] := 1.0;
   DATA[1326,4] := 262.5609;
   DATA[1326,5] := 8.464369;
   DATA[1326,6] := 317.9185;
   DATA[1326,8] := 1.0;
   DATA[1326,9] := 1.0;
   DATA[1326,10] := 1.0;
   DATA[1326,11] := 0.9091491;
   DATA[1326,12] := 0.000384332;
   DATA[1326,13] := 1010.959;
   DATA[1326,14] := 1.0;
   DATA[1326,15] := 1.0;
   DATA[1326,16] := 1.0;
   DATA[1326,18] := 1.0;
   DATA[1326,19] := 1.0;
   DATA[1326,20] := 148.808;
   DATA[1326,21] := 154.0118;
   DATA[1326,22] := 1.713517;
   DATA[1326,23] := 798.6029;
   DATA[1326,24] := 2.0;
   DATA[1326,25] := 2.0;
   DATA[1326,26] := 7.87798;
   DATA[1326,27] := 142.9633;
   DATA[1326,28] := 263.0095;
   DATA[1326,29] := 12.07383;
   DATA[1326,30] := 1.723789;
   DATA[1326,31] := 1.267837;
   DATA[1326,32] := 0.736421;
   DATA[1326,33] := 0.3081703;
   DATA[1326,34] := 2.0;
   DATA[1326,35] := 249.7917;
   DATA[1326,36] := 1.617916;
   DATA[1326,37] := 188.6856;
   DATA[1326,38] := 0.000128152;
   DATA[1326,39] := 1.0;
   DATA[1327,1] := 813.8275;
   DATA[1327,2] := 1.0;
   DATA[1327,3] := 1.0;
   DATA[1327,4] := 262.5609;
   DATA[1327,5] := 8.464369;
   DATA[1327,6] := 317.9185;
   DATA[1327,8] := 1.0;
   DATA[1327,9] := 1.0;
   DATA[1327,10] := 1.0;
   DATA[1327,11] := 0.768295;
   DATA[1327,13] := 1010.678;
   DATA[1327,14] := 1.0;
   DATA[1327,15] := 1.0;
   DATA[1327,16] := 1.0;
   DATA[1327,18] := 1.0;
   DATA[1327,19] := 1.0;
   DATA[1327,20] := 148.808;
   DATA[1327,21] := 154.0118;
   DATA[1327,22] := 1.713517;
   DATA[1327,23] := 798.4106;
   DATA[1327,24] := 2.0;
   DATA[1327,25] := 2.0;
   DATA[1327,26] := 7.87798;
   DATA[1327,27] := 142.9633;
   DATA[1327,28] := 263.0095;
   DATA[1327,29] := 12.07383;
   DATA[1327,30] := 1.722763;
   DATA[1327,31] := 1.266299;
   DATA[1327,32] := 0.7348846;
   DATA[1327,33] := 0.3081703;
   DATA[1327,34] := 2.0;
   DATA[1327,35] := 249.9199;
   DATA[1327,36] := 1.617916;
   DATA[1327,37] := 188.7817;
   DATA[1327,38] := 0.000128152;
   DATA[1327,39] := 1.0;
   DATA[1328,1] := 814.1807;
   DATA[1328,2] := 1.0;
   DATA[1328,3] := 1.0;
   DATA[1328,4] := 262.5609;
   DATA[1328,5] := 8.464369;
   DATA[1328,6] := 317.9185;
   DATA[1328,8] := 1.0;
   DATA[1328,9] := 1.0;
   DATA[1328,10] := 1.0;
   DATA[1328,11] := 0.7490876;
   DATA[1328,13] := 1010.919;
   DATA[1328,14] := 1.0;
   DATA[1328,15] := 1.0;
   DATA[1328,16] := 1.0;
   DATA[1328,18] := 1.0;
   DATA[1328,19] := 1.0;
   DATA[1328,20] := 148.808;
   DATA[1328,21] := 154.0118;
   DATA[1328,22] := 1.713517;
   DATA[1328,23] := 798.103;
   DATA[1328,24] := 2.0;
   DATA[1328,25] := 2.0;
   DATA[1328,26] := 7.87798;
   DATA[1328,27] := 142.9633;
   DATA[1328,28] := 263.0095;
   DATA[1328,29] := 12.07383;
   DATA[1328,30] := 1.722123;
   DATA[1328,31] := 1.272192;
   DATA[1328,32] := 0.7348846;
   DATA[1328,33] := 0.3082983;
   DATA[1328,34] := 2.0;
   DATA[1328,35] := 250.016;
   DATA[1328,36] := 1.746067;
   DATA[1328,37] := 188.8939;
   DATA[1328,38] := 0.000128152;
   DATA[1328,39] := 1.0;
   DATA[1329,1] := 814.4162;
   DATA[1329,2] := 1.0;
   DATA[1329,3] := 1.0;
   DATA[1329,4] := 262.5609;
   DATA[1329,5] := 8.464369;
   DATA[1329,6] := 317.9185;
   DATA[1329,8] := 1.0;
   DATA[1329,9] := 1.0;
   DATA[1329,10] := 1.0;
   DATA[1329,11] := 0.7907037;
   DATA[1329,13] := 1010.758;
   DATA[1329,14] := 1.0;
   DATA[1329,15] := 1.0;
   DATA[1329,16] := 1.0;
   DATA[1329,17] := 2.0;
   DATA[1329,18] := 1.0;
   DATA[1329,19] := 2.0;
   DATA[1329,20] := 148.808;
   DATA[1329,21] := 153.9862;
   DATA[1329,22] := 1.711723;
   DATA[1329,23] := 798.0646;
   DATA[1329,24] := 2.0;
   DATA[1329,25] := 2.0;
   DATA[1329,26] := 7.87798;
   DATA[1329,27] := 142.9633;
   DATA[1329,28] := 263.0095;
   DATA[1329,29] := 12.07383;
   DATA[1329,30] := 1.721482;
   DATA[1329,31] := 1.282183;
   DATA[1329,32] := 0.7348846;
   DATA[1329,33] := 0.3086827;
   DATA[1329,34] := 2.0;
   DATA[1329,35] := 250.016;
   DATA[1329,36] := 1.746067;
   DATA[1329,37] := 188.8939;
   DATA[1329,38] := 0.000128152;
   DATA[1329,39] := 1.0;
   DATA[1330,1] := 814.8873;
   DATA[1330,2] := 1.0;
   DATA[1330,3] := 1.0;
   DATA[1330,4] := 262.5609;
   DATA[1330,5] := 8.464048;
   DATA[1330,6] := 317.9185;
   DATA[1330,8] := 1.0;
   DATA[1330,9] := 1.0;
   DATA[1330,10] := 1.0;
   DATA[1330,11] := 1.174851;
   DATA[1330,13] := 1010.718;
   DATA[1330,14] := 1.0;
   DATA[1330,15] := 1.0;
   DATA[1330,16] := 1.0;
   DATA[1330,17] := 2.0;
   DATA[1330,18] := 1.0;
   DATA[1330,19] := 2.0;
   DATA[1330,20] := 148.808;
   DATA[1330,21] := 153.8836;
   DATA[1330,22] := 1.711466;
   DATA[1330,23] := 798.2953;
   DATA[1330,24] := 2.0;
   DATA[1330,25] := 2.0;
   DATA[1330,26] := 7.87798;
   DATA[1330,27] := 142.9633;
   DATA[1330,28] := 263.0095;
   DATA[1330,29] := 12.07383;
   DATA[1330,30] := 1.721482;
   DATA[1330,31] := 1.277059;
   DATA[1330,32] := 0.7348846;
   DATA[1330,33] := 0.3086827;
   DATA[1330,34] := 2.0;
   DATA[1330,35] := 250.016;
   DATA[1330,36] := 1.746067;
   DATA[1330,37] := 188.8939;
   DATA[1330,38] := 0.000128152;
   DATA[1330,39] := 1.0;
   DATA[1331,1] := 815.005;
   DATA[1331,2] := 1.0;
   DATA[1331,3] := 1.0;
   DATA[1331,4] := 262.5609;
   DATA[1331,5] := 8.460844;
   DATA[1331,6] := 317.9185;
   DATA[1331,8] := 1.0;
   DATA[1331,9] := 1.0;
   DATA[1331,10] := 1.0;
   DATA[1331,11] := 1.898329;
   DATA[1331,12] := 0.000512443;
   DATA[1331,13] := 1010.438;
   DATA[1331,14] := 1.0;
   DATA[1331,15] := 1.0;
   DATA[1331,16] := 1.0;
   DATA[1331,17] := 2.0;
   DATA[1331,18] := 1.0;
   DATA[1331,19] := 2.0;
   DATA[1331,20] := 148.808;
   DATA[1331,21] := 153.8836;
   DATA[1331,22] := 1.711466;
   DATA[1331,23] := 797.8723;
   DATA[1331,24] := 2.0;
   DATA[1331,25] := 2.0;
   DATA[1331,26] := 7.87798;
   DATA[1331,27] := 142.9633;
   DATA[1331,28] := 263.0095;
   DATA[1331,29] := 12.07383;
   DATA[1331,30] := 1.721482;
   DATA[1331,31] := 1.283464;
   DATA[1331,32] := 0.7348846;
   DATA[1331,33] := 0.3086827;
   DATA[1331,34] := 2.0;
   DATA[1331,35] := 250.1442;
   DATA[1331,36] := 1.746067;
   DATA[1331,37] := 188.8939;
   DATA[1331,38] := 0.000128152;
   DATA[1331,39] := 1.0;
   DATA[1332,1] := 814.691;
   DATA[1332,2] := 1.0;
   DATA[1332,3] := 1.0;
   DATA[1332,4] := 262.5609;
   DATA[1332,5] := 8.460844;
   DATA[1332,6] := 317.9185;
   DATA[1332,8] := 1.0;
   DATA[1332,9] := 1.0;
   DATA[1332,10] := 1.0;
   DATA[1332,11] := 2.8651;
   DATA[1332,12] := 0.03625532;
   DATA[1332,13] := 1010.678;
   DATA[1332,14] := 1.0;
   DATA[1332,15] := 1.0;
   DATA[1332,16] := 1.0;
   DATA[1332,17] := 2.0;
   DATA[1332,18] := 1.0;
   DATA[1332,19] := 2.0;
   DATA[1332,20] := 148.808;
   DATA[1332,21] := 153.8836;
   DATA[1332,22] := 1.711466;
   DATA[1332,23] := 797.6801;
   DATA[1332,24] := 2.0;
   DATA[1332,25] := 2.0;
   DATA[1332,26] := 7.87798;
   DATA[1332,27] := 142.9633;
   DATA[1332,28] := 263.0095;
   DATA[1332,29] := 12.07383;
   DATA[1332,30] := 1.723661;
   DATA[1332,31] := 1.283464;
   DATA[1332,32] := 0.7348846;
   DATA[1332,33] := 0.3086827;
   DATA[1332,34] := 2.0;
   DATA[1332,35] := 250.1602;
   DATA[1332,36] := 1.681991;
   DATA[1332,37] := 189.1342;
   DATA[1332,38] := 0.000128152;
   DATA[1332,39] := 1.0;
   DATA[1333,1] := 814.7695;
   DATA[1333,2] := 1.0;
   DATA[1333,3] := 1.0;
   DATA[1333,4] := 262.5609;
   DATA[1333,5] := 8.460844;
   DATA[1333,6] := 317.9185;
   DATA[1333,8] := 1.0;
   DATA[1333,9] := 1.0;
   DATA[1333,10] := 1.0;
   DATA[1333,11] := 3.969524;
   DATA[1333,12] := 0.2099734;
   DATA[1333,13] := 1010.718;
   DATA[1333,14] := 1.0;
   DATA[1333,15] := 1.0;
   DATA[1333,16] := 1.0;
   DATA[1333,17] := 2.0;
   DATA[1333,18] := 1.0;
   DATA[1333,19] := 2.0;
   DATA[1333,20] := 148.808;
   DATA[1333,21] := 153.8836;
   DATA[1333,22] := 1.714029;
   DATA[1333,23] := 797.334;
   DATA[1333,24] := 2.0;
   DATA[1333,25] := 2.0;
   DATA[1333,26] := 7.87798;
   DATA[1333,27] := 142.9633;
   DATA[1333,28] := 263.0095;
   DATA[1333,29] := 12.07383;
   DATA[1333,30] := 1.723661;
   DATA[1333,31] := 1.283464;
   DATA[1333,32] := 0.7348846;
   DATA[1333,33] := 0.3086827;
   DATA[1333,34] := 2.0;
   DATA[1333,35] := 250.2563;
   DATA[1333,36] := 1.681991;
   DATA[1333,37] := 189.1342;
   DATA[1333,38] := 0.000128152;
   DATA[1333,39] := 1.0;
   DATA[1334,1] := 814.8873;
   DATA[1334,2] := 1.0;
   DATA[1334,3] := 1.0;
   DATA[1334,4] := 262.5609;
   DATA[1334,5] := 8.460844;
   DATA[1334,6] := 317.9185;
   DATA[1334,8] := 1.0;
   DATA[1334,9] := 1.0;
   DATA[1334,10] := 1.0;
   DATA[1334,11] := 5.109162;
   DATA[1334,12] := 0.4691413;
   DATA[1334,13] := 1010.758;
   DATA[1334,14] := 1.0;
   DATA[1334,15] := 1.0;
   DATA[1334,16] := 1.0;
   DATA[1334,17] := 2.0;
   DATA[1334,18] := 1.0;
   DATA[1334,19] := 2.0;
   DATA[1334,20] := 148.808;
   DATA[1334,21] := 153.8836;
   DATA[1334,22] := 1.71467;
   DATA[1334,23] := 796.9495;
   DATA[1334,24] := 2.0;
   DATA[1334,25] := 2.0;
   DATA[1334,26] := 7.87798;
   DATA[1334,27] := 142.9633;
   DATA[1334,28] := 263.0095;
   DATA[1334,29] := 12.07383;
   DATA[1334,30] := 1.723661;
   DATA[1334,31] := 1.290637;
   DATA[1334,32] := 0.7353967;
   DATA[1334,33] := 0.3083624;
   DATA[1334,34] := 2.0;
   DATA[1334,35] := 250.3204;
   DATA[1334,36] := 1.681991;
   DATA[1334,37] := 189.1342;
   DATA[1334,38] := 0.000128152;
   DATA[1334,39] := 1.0;
   DATA[1335,1] := 814.9658;
   DATA[1335,2] := 1.0;
   DATA[1335,3] := 1.0;
   DATA[1335,4] := 262.5609;
   DATA[1335,5] := 8.460844;
   DATA[1335,6] := 317.9185;
   DATA[1335,8] := 1.0;
   DATA[1335,9] := 1.0;
   DATA[1335,10] := 1.0;
   DATA[1335,11] := 6.152762;
   DATA[1335,12] := 0.8364347;
   DATA[1335,13] := 1010.678;
   DATA[1335,14] := 1.0;
   DATA[1335,15] := 1.0;
   DATA[1335,16] := 1.0;
   DATA[1335,17] := 2.0;
   DATA[1335,18] := 1.0;
   DATA[1335,19] := 2.0;
   DATA[1335,20] := 148.808;
   DATA[1335,21] := 153.8836;
   DATA[1335,22] := 1.715311;
   DATA[1335,23] := 796.1805;
   DATA[1335,24] := 2.0;
   DATA[1335,25] := 2.0;
   DATA[1335,26] := 7.87798;
   DATA[1335,27] := 142.9633;
   DATA[1335,28] := 263.0095;
   DATA[1335,29] := 12.07383;
   DATA[1335,30] := 1.723661;
   DATA[1335,31] := 1.291789;
   DATA[1335,32] := 0.7353967;
   DATA[1335,33] := 0.3083624;
   DATA[1335,34] := 2.0;
   DATA[1335,35] := 250.3204;
   DATA[1335,36] := 1.681991;
   DATA[1335,37] := 189.1342;
   DATA[1335,38] := 0.000128152;
   DATA[1335,39] := 1.0;
   DATA[1336,1] := 814.8873;
   DATA[1336,2] := 1.0;
   DATA[1336,3] := 1.0;
   DATA[1336,4] := 262.5609;
   DATA[1336,5] := 8.460844;
   DATA[1336,6] := 317.9185;
   DATA[1336,8] := 1.0;
   DATA[1336,9] := 1.0;
   DATA[1336,10] := 1.0;
   DATA[1336,11] := 7.193162;
   DATA[1336,12] := 1.207699;
   DATA[1336,13] := 1010.879;
   DATA[1336,14] := 1.0;
   DATA[1336,15] := 1.0;
   DATA[1336,16] := 1.0;
   DATA[1336,17] := 2.0;
   DATA[1336,18] := 1.0;
   DATA[1336,19] := 2.0;
   DATA[1336,20] := 148.808;
   DATA[1336,21] := 153.8836;
   DATA[1336,22] := 1.715311;
   DATA[1336,23] := 795.9113;
   DATA[1336,24] := 2.0;
   DATA[1336,25] := 2.0;
   DATA[1336,26] := 7.87798;
   DATA[1336,27] := 142.9633;
   DATA[1336,28] := 263.0095;
   DATA[1336,29] := 12.07383;
   DATA[1336,30] := 1.723661;
   DATA[1336,31] := 1.293198;
   DATA[1336,32] := 0.7353967;
   DATA[1336,33] := 0.3083624;
   DATA[1336,34] := 2.0;
   DATA[1336,35] := 250.3204;
   DATA[1336,36] := 1.681991;
   DATA[1336,37] := 189.1342;
   DATA[1336,38] := 0.000128152;
   DATA[1336,39] := 1.0;
   DATA[1337,1] := 814.4948;
   DATA[1337,2] := 1.0;
   DATA[1337,3] := 1.0;
   DATA[1337,4] := 262.5609;
   DATA[1337,5] := 8.460844;
   DATA[1337,6] := 317.9185;
   DATA[1337,8] := 1.0;
   DATA[1337,9] := 1.0;
   DATA[1337,10] := 1.0;
   DATA[1337,11] := 7.900634;
   DATA[1337,12] := 1.584985;
   DATA[1337,13] := 1010.438;
   DATA[1337,14] := 1.0;
   DATA[1337,15] := 1.0;
   DATA[1337,16] := 1.0;
   DATA[1337,17] := 2.0;
   DATA[1337,18] := 1.0;
   DATA[1337,19] := 2.0;
   DATA[1337,20] := 148.808;
   DATA[1337,21] := 153.8836;
   DATA[1337,22] := 1.715311;
   DATA[1337,23] := 795.5268;
   DATA[1337,24] := 2.0;
   DATA[1337,25] := 2.0;
   DATA[1337,26] := 7.87798;
   DATA[1337,27] := 142.9633;
   DATA[1337,28] := 263.0095;
   DATA[1337,29] := 12.07383;
   DATA[1337,30] := 1.723661;
   DATA[1337,31] := 1.300756;
   DATA[1337,32] := 0.7353967;
   DATA[1337,33] := 0.3083624;
   DATA[1337,34] := 2.0;
   DATA[1337,35] := 250.3204;
   DATA[1337,36] := 1.681991;
   DATA[1337,37] := 189.1342;
   DATA[1337,38] := 0.000128152;
   DATA[1337,39] := 1.0;
   DATA[1338,1] := 814.22;
   DATA[1338,2] := 1.0;
   DATA[1338,3] := 1.0;
   DATA[1338,4] := 262.5609;
   DATA[1338,5] := 8.460844;
   DATA[1338,6] := 317.9185;
   DATA[1338,8] := 1.0;
   DATA[1338,9] := 1.0;
   DATA[1338,10] := 1.0;
   DATA[1338,11] := 8.422434;
   DATA[1338,12] := 1.850943;
   DATA[1338,13] := 1010.638;
   DATA[1338,14] := 1.0;
   DATA[1338,15] := 1.0;
   DATA[1338,16] := 1.0;
   DATA[1338,17] := 2.0;
   DATA[1338,18] := 1.0;
   DATA[1338,19] := 2.0;
   DATA[1338,20] := 148.808;
   DATA[1338,21] := 153.8836;
   DATA[1338,22] := 1.715311;
   DATA[1338,23] := 795.0654;
   DATA[1338,24] := 2.0;
   DATA[1338,25] := 2.0;
   DATA[1338,26] := 7.87798;
   DATA[1338,27] := 142.9633;
   DATA[1338,28] := 263.0095;
   DATA[1338,29] := 12.07383;
   DATA[1338,30] := 1.725583;
   DATA[1338,31] := 1.290893;
   DATA[1338,32] := 0.7353967;
   DATA[1338,33] := 0.3083624;
   DATA[1338,34] := 2.0;
   DATA[1338,35] := 250.3204;
   DATA[1338,36] := 1.681991;
   DATA[1338,37] := 189.1342;
   DATA[1338,38] := 0.000128152;
   DATA[1338,39] := 1.0;
   DATA[1339,1] := 814.22;
   DATA[1339,2] := 1.0;
   DATA[1339,3] := 1.0;
   DATA[1339,4] := 262.5609;
   DATA[1339,5] := 8.460844;
   DATA[1339,6] := 317.9185;
   DATA[1339,8] := 1.0;
   DATA[1339,9] := 1.0;
   DATA[1339,10] := 1.0;
   DATA[1339,11] := 8.422434;
   DATA[1339,12] := 1.850943;
   DATA[1339,13] := 1010.638;
   DATA[1339,14] := 1.0;
   DATA[1339,15] := 1.0;
   DATA[1339,16] := 1.0;
   DATA[1339,17] := 2.0;
   DATA[1339,18] := 1.0;
   DATA[1339,19] := 2.0;
   DATA[1339,20] := 148.808;
   DATA[1339,21] := 153.8836;
   DATA[1339,22] := 1.715311;
   DATA[1339,23] := 795.0654;
   DATA[1339,24] := 2.0;
   DATA[1339,25] := 2.0;
   DATA[1339,26] := 7.87798;
   DATA[1339,27] := 142.9633;
   DATA[1339,28] := 263.0095;
   DATA[1339,29] := 12.07383;
   DATA[1339,30] := 1.725583;
   DATA[1339,31] := 1.290893;
   DATA[1339,32] := 0.7353967;
   DATA[1339,33] := 0.3083624;
   DATA[1339,34] := 2.0;
   DATA[1339,35] := 250.3204;
   DATA[1339,36] := 1.681991;
   DATA[1339,37] := 189.1342;
   DATA[1339,38] := 0.000128152;
   DATA[1339,39] := 1.0;
   DATA[1340,1] := 814.3377;
   DATA[1340,2] := 1.0;
   DATA[1340,3] := 1.0;
   DATA[1340,4] := 262.5609;
   DATA[1340,5] := 8.460844;
   DATA[1340,6] := 317.9185;
   DATA[1340,8] := 1.0;
   DATA[1340,9] := 1.0;
   DATA[1340,10] := 1.0;
   DATA[1340,11] := 8.947435;
   DATA[1340,12] := 2.017359;
   DATA[1340,13] := 1010.278;
   DATA[1340,14] := 1.0;
   DATA[1340,15] := 1.0;
   DATA[1340,16] := 1.0;
   DATA[1340,17] := 2.0;
   DATA[1340,18] := 1.0;
   DATA[1340,19] := 2.0;
   DATA[1340,20] := 148.808;
   DATA[1340,21] := 153.8836;
   DATA[1340,22] := 1.715311;
   DATA[1340,23] := 795.1807;
   DATA[1340,24] := 2.0;
   DATA[1340,25] := 2.0;
   DATA[1340,26] := 7.87798;
   DATA[1340,27] := 142.9633;
   DATA[1340,28] := 263.0095;
   DATA[1340,29] := 12.30454;
   DATA[1340,30] := 1.725583;
   DATA[1340,31] := 1.281798;
   DATA[1340,32] := 0.7353967;
   DATA[1340,33] := 0.3083624;
   DATA[1340,34] := 2.0;
   DATA[1340,35] := 250.3204;
   DATA[1340,36] := 1.681991;
   DATA[1340,37] := 189.1342;
   DATA[1340,38] := 0.000128152;
   DATA[1340,39] := 1.0;
   DATA[1341,1] := 814.377;
   DATA[1341,2] := 1.0;
   DATA[1341,3] := 1.0;
   DATA[1341,4] := 262.5609;
   DATA[1341,5] := 8.460844;
   DATA[1341,6] := 317.9185;
   DATA[1341,8] := 1.0;
   DATA[1341,9] := 1.0;
   DATA[1341,10] := 1.0;
   DATA[1341,11] := 9.357193;
   DATA[1341,12] := 2.117157;
   DATA[1341,13] := 1010.078;
   DATA[1341,14] := 1.0;
   DATA[1341,15] := 1.0;
   DATA[1341,16] := 1.0;
   DATA[1341,17] := 2.0;
   DATA[1341,18] := 1.0;
   DATA[1341,19] := 2.0;
   DATA[1341,20] := 148.808;
   DATA[1341,21] := 153.8836;
   DATA[1341,22] := 1.716208;
   DATA[1341,23] := 794.9885;
   DATA[1341,24] := 2.0;
   DATA[1341,25] := 2.0;
   DATA[1341,26] := 7.87798;
   DATA[1341,27] := 142.9633;
   DATA[1341,28] := 263.0095;
   DATA[1341,29] := 12.30454;
   DATA[1341,30] := 1.725455;
   DATA[1341,31] := 1.281286;
   DATA[1341,32] := 0.7353967;
   DATA[1341,33] := 0.3083624;
   DATA[1341,34] := 2.0;
   DATA[1341,35] := 250.1122;
   DATA[1341,36] := 1.681991;
   DATA[1341,37] := 189.1342;
   DATA[1341,38] := 0.000128152;
   DATA[1341,39] := 1.0;
   DATA[1342,1] := 814.22;
   DATA[1342,2] := 1.0;
   DATA[1342,3] := 1.0;
   DATA[1342,4] := 262.5609;
   DATA[1342,5] := 8.460844;
   DATA[1342,6] := 317.9185;
   DATA[1342,8] := 1.0;
   DATA[1342,9] := 1.0;
   DATA[1342,10] := 1.0;
   DATA[1342,11] := 9.45323;
   DATA[1342,12] := 2.175704;
   DATA[1342,13] := 1009.717;
   DATA[1342,14] := 1.0;
   DATA[1342,15] := 1.0;
   DATA[1342,16] := 1.0;
   DATA[1342,17] := 2.0;
   DATA[1342,18] := 1.0;
   DATA[1342,19] := 2.0;
   DATA[1342,20] := 148.808;
   DATA[1342,21] := 153.8836;
   DATA[1342,22] := 1.716208;
   DATA[1342,23] := 794.2963;
   DATA[1342,24] := 2.0;
   DATA[1342,25] := 2.0;
   DATA[1342,26] := 7.87798;
   DATA[1342,27] := 142.9633;
   DATA[1342,28] := 263.0095;
   DATA[1342,29] := 12.30454;
   DATA[1342,30] := 1.724686;
   DATA[1342,31] := 1.281286;
   DATA[1342,32] := 0.7353967;
   DATA[1342,33] := 0.3083624;
   DATA[1342,34] := 2.0;
   DATA[1342,35] := 250.0961;
   DATA[1342,36] := 1.681991;
   DATA[1342,37] := 189.1342;
   DATA[1342,38] := 0.000128152;
   DATA[1342,39] := 1.0;
   DATA[1343,1] := 814.6125;
   DATA[1343,2] := 1.0;
   DATA[1343,3] := 1.0;
   DATA[1343,4] := 262.5609;
   DATA[1343,5] := 8.462446;
   DATA[1343,6] := 317.9185;
   DATA[1343,8] := 1.0;
   DATA[1343,9] := 1.0;
   DATA[1343,10] := 1.0;
   DATA[1343,11] := 9.526858;
   DATA[1343,12] := 2.209525;
   DATA[1343,13] := 1009.557;
   DATA[1343,14] := 1.0;
   DATA[1343,15] := 1.0;
   DATA[1343,16] := 1.0;
   DATA[1343,17] := 2.0;
   DATA[1343,18] := 1.0;
   DATA[1343,19] := 2.0;
   DATA[1343,20] := 148.808;
   DATA[1343,21] := 153.8836;
   DATA[1343,22] := 1.716208;
   DATA[1343,23] := 793.758;
   DATA[1343,24] := 2.0;
   DATA[1343,25] := 2.0;
   DATA[1343,26] := 7.87798;
   DATA[1343,27] := 142.9633;
   DATA[1343,28] := 263.0095;
   DATA[1343,29] := 12.07383;
   DATA[1343,30] := 1.724686;
   DATA[1343,31] := 1.281286;
   DATA[1343,32] := 0.7353967;
   DATA[1343,33] := 0.3083624;
   DATA[1343,34] := 2.0;
   DATA[1343,35] := 250.0961;
   DATA[1343,36] := 1.681991;
   DATA[1343,37] := 189.0541;
   DATA[1343,38] := 0.000128152;
   DATA[1343,39] := 1.0;
   DATA[1344,1] := 814.7695;
   DATA[1344,2] := 1.0;
   DATA[1344,3] := 1.0;
   DATA[1344,4] := 262.5609;
   DATA[1344,5] := 8.462446;
   DATA[1344,6] := 317.9185;
   DATA[1344,8] := 1.0;
   DATA[1344,9] := 1.0;
   DATA[1344,10] := 1.0;
   DATA[1344,11] := 9.526858;
   DATA[1344,12] := 2.230023;
   DATA[1344,13] := 1009.156;
   DATA[1344,14] := 1.0;
   DATA[1344,15] := 1.0;
   DATA[1344,16] := 1.0;
   DATA[1344,17] := 2.0;
   DATA[1344,18] := 1.0;
   DATA[1344,19] := 2.0;
   DATA[1344,20] := 148.808;
   DATA[1344,21] := 153.8836;
   DATA[1344,22] := 1.716208;
   DATA[1344,23] := 793.7195;
   DATA[1344,24] := 2.0;
   DATA[1344,25] := 2.0;
   DATA[1344,26] := 7.87798;
   DATA[1344,27] := 142.989;
   DATA[1344,28] := 263.0095;
   DATA[1344,29] := 11.95847;
   DATA[1344,30] := 1.724814;
   DATA[1344,31] := 1.281286;
   DATA[1344,32] := 0.7353967;
   DATA[1344,33] := 0.3083624;
   DATA[1344,34] := 2.0;
   DATA[1344,35] := 250.0961;
   DATA[1344,36] := 1.681991;
   DATA[1344,37] := 189.0541;
   DATA[1344,38] := 0.000128152;
   DATA[1344,39] := 1.0;
   DATA[1345,1] := 814.534;
   DATA[1345,2] := 1.0;
   DATA[1345,3] := 1.0;
   DATA[1345,4] := 262.5609;
   DATA[1345,5] := 8.462446;
   DATA[1345,6] := 317.9185;
   DATA[1345,8] := 1.0;
   DATA[1345,9] := 1.0;
   DATA[1345,10] := 1.0;
   DATA[1345,11] := 9.55887;
   DATA[1345,12] := 2.236044;
   DATA[1345,13] := 1009.236;
   DATA[1345,14] := 1.0;
   DATA[1345,15] := 1.0;
   DATA[1345,16] := 1.0;
   DATA[1345,17] := 2.0;
   DATA[1345,18] := 1.0;
   DATA[1345,19] := 2.0;
   DATA[1345,20] := 148.808;
   DATA[1345,21] := 153.8836;
   DATA[1345,22] := 1.716208;
   DATA[1345,23] := 793.4504;
   DATA[1345,24] := 2.0;
   DATA[1345,25] := 2.0;
   DATA[1345,26] := 7.87798;
   DATA[1345,27] := 143.0403;
   DATA[1345,28] := 263.1056;
   DATA[1345,29] := 11.95847;
   DATA[1345,30] := 1.726865;
   DATA[1345,31] := 1.269502;
   DATA[1345,32] := 0.7353967;
   DATA[1345,33] := 0.3083624;
   DATA[1345,34] := 2.0;
   DATA[1345,35] := 250.2724;
   DATA[1345,36] := 1.681991;
   DATA[1345,37] := 189.0541;
   DATA[1345,38] := 0.000128152;
   DATA[1345,39] := 1.0;
   DATA[1346,1] := 814.534;
   DATA[1346,2] := 1.0;
   DATA[1346,3] := 1.0;
   DATA[1346,4] := 262.5609;
   DATA[1346,5] := 8.462446;
   DATA[1346,6] := 317.9185;
   DATA[1346,8] := 1.0;
   DATA[1346,9] := 1.0;
   DATA[1346,10] := 1.0;
   DATA[1346,11] := 9.491645;
   DATA[1346,12] := 2.231304;
   DATA[1346,13] := 1008.515;
   DATA[1346,14] := 1.0;
   DATA[1346,15] := 1.0;
   DATA[1346,16] := 1.0;
   DATA[1346,17] := 2.0;
   DATA[1346,18] := 1.0;
   DATA[1346,19] := 2.0;
   DATA[1346,20] := 148.808;
   DATA[1346,21] := 153.8836;
   DATA[1346,22] := 1.716208;
   DATA[1346,23] := 793.2197;
   DATA[1346,24] := 2.0;
   DATA[1346,25] := 2.0;
   DATA[1346,26] := 7.87798;
   DATA[1346,27] := 143.0403;
   DATA[1346,28] := 263.1056;
   DATA[1346,29] := 11.95847;
   DATA[1346,30] := 1.727378;
   DATA[1346,31] := 1.262073;
   DATA[1346,32] := 0.7353967;
   DATA[1346,33] := 0.3083624;
   DATA[1346,34] := 2.0;
   DATA[1346,35] := 250.2724;
   DATA[1346,36] := 1.681991;
   DATA[1346,37] := 189.0541;
   DATA[1346,38] := 0.000128152;
   DATA[1346,39] := 1.0;
   DATA[1347,1] := 814.7302;
   DATA[1347,2] := 1.0;
   DATA[1347,3] := 1.0;
   DATA[1347,4] := 262.5609;
   DATA[1347,5] := 8.462446;
   DATA[1347,6] := 317.9185;
   DATA[1347,8] := 1.0;
   DATA[1347,9] := 1.0;
   DATA[1347,10] := 1.0;
   DATA[1347,11] := 9.450028;
   DATA[1347,12] := 2.228613;
   DATA[1347,13] := 1008.355;
   DATA[1347,14] := 1.0;
   DATA[1347,15] := 1.0;
   DATA[1347,16] := 1.0;
   DATA[1347,17] := 2.0;
   DATA[1347,18] := 1.0;
   DATA[1347,19] := 2.0;
   DATA[1347,20] := 148.808;
   DATA[1347,21] := 153.8836;
   DATA[1347,22] := 1.716592;
   DATA[1347,23] := 793.1812;
   DATA[1347,24] := 2.0;
   DATA[1347,25] := 2.0;
   DATA[1347,26] := 7.87798;
   DATA[1347,27] := 143.0403;
   DATA[1347,28] := 263.1056;
   DATA[1347,29] := 12.30454;
   DATA[1347,30] := 1.727378;
   DATA[1347,31] := 1.273857;
   DATA[1347,32] := 0.7353967;
   DATA[1347,33] := 0.3083624;
   DATA[1347,34] := 2.0;
   DATA[1347,35] := 250.2724;
   DATA[1347,36] := 1.681991;
   DATA[1347,37] := 189.0541;
   DATA[1347,38] := 0.000128152;
   DATA[1347,39] := 1.0;
   DATA[1348,1] := 814.6125;
   DATA[1348,2] := 1.0;
   DATA[1348,3] := 1.0;
   DATA[1348,4] := 262.5609;
   DATA[1348,5] := 8.462446;
   DATA[1348,6] := 317.9185;
   DATA[1348,8] := 1.0;
   DATA[1348,9] := 1.0;
   DATA[1348,10] := 1.0;
   DATA[1348,11] := 9.42762;
   DATA[1348,12] := 2.227076;
   DATA[1348,13] := 1007.915;
   DATA[1348,14] := 1.0;
   DATA[1348,15] := 1.0;
   DATA[1348,16] := 1.0;
   DATA[1348,17] := 2.0;
   DATA[1348,18] := 1.0;
   DATA[1348,19] := 2.0;
   DATA[1348,20] := 148.808;
   DATA[1348,21] := 153.8836;
   DATA[1348,22] := 1.717489;
   DATA[1348,23] := 792.7582;
   DATA[1348,24] := 2.0;
   DATA[1348,25] := 2.0;
   DATA[1348,26] := 7.87798;
   DATA[1348,27] := 143.0403;
   DATA[1348,28] := 263.1056;
   DATA[1348,29] := 12.30454;
   DATA[1348,30] := 1.727378;
   DATA[1348,31] := 1.282439;
   DATA[1348,32] := 0.7353967;
   DATA[1348,33] := 0.3083624;
   DATA[1348,34] := 2.0;
   DATA[1348,35] := 250.3525;
   DATA[1348,36] := 1.681991;
   DATA[1348,37] := 189.0541;
   DATA[1348,38] := 0.000128152;
   DATA[1348,39] := 1.0;
   DATA[1349,1] := 814.6125;
   DATA[1349,2] := 1.0;
   DATA[1349,3] := 1.0;
   DATA[1349,4] := 262.5609;
   DATA[1349,5] := 8.462446;
   DATA[1349,6] := 317.9185;
   DATA[1349,8] := 1.0;
   DATA[1349,9] := 1.0;
   DATA[1349,10] := 1.0;
   DATA[1349,11] := 9.42762;
   DATA[1349,12] := 2.225795;
   DATA[1349,13] := 1007.434;
   DATA[1349,14] := 1.0;
   DATA[1349,15] := 1.0;
   DATA[1349,16] := 1.0;
   DATA[1349,17] := 2.0;
   DATA[1349,18] := 1.0;
   DATA[1349,19] := 2.0;
   DATA[1349,20] := 148.808;
   DATA[1349,21] := 153.8836;
   DATA[1349,22] := 1.717489;
   DATA[1349,23] := 792.4122;
   DATA[1349,24] := 2.0;
   DATA[1349,25] := 2.0;
   DATA[1349,26] := 7.87798;
   DATA[1349,27] := 143.0403;
   DATA[1349,28] := 263.1056;
   DATA[1349,29] := 12.30454;
   DATA[1349,30] := 1.727378;
   DATA[1349,31] := 1.283848;
   DATA[1349,32] := 0.7353967;
   DATA[1349,33] := 0.3083624;
   DATA[1349,34] := 2.0;
   DATA[1349,35] := 250.3525;
   DATA[1349,36] := 1.681991;
   DATA[1349,37] := 189.0541;
   DATA[1349,38] := 0.000128152;
   DATA[1349,39] := 1.0;
   DATA[1350,1] := 814.4162;
   DATA[1350,2] := 1.0;
   DATA[1350,3] := 1.0;
   DATA[1350,4] := 262.5609;
   DATA[1350,5] := 8.462446;
   DATA[1350,6] := 317.9185;
   DATA[1350,8] := 1.0;
   DATA[1350,9] := 1.0;
   DATA[1350,10] := 1.0;
   DATA[1350,11] := 9.42762;
   DATA[1350,12] := 2.225667;
   DATA[1350,13] := 1006.353;
   DATA[1350,14] := 1.0;
   DATA[1350,15] := 1.0;
   DATA[1350,16] := 1.0;
   DATA[1350,17] := 2.0;
   DATA[1350,18] := 1.0;
   DATA[1350,19] := 2.0;
   DATA[1350,20] := 148.808;
   DATA[1350,21] := 153.8836;
   DATA[1350,22] := 1.717489;
   DATA[1350,23] := 791.9893;
   DATA[1350,24] := 2.0;
   DATA[1350,25] := 2.0;
   DATA[1350,26] := 7.87798;
   DATA[1350,27] := 143.0403;
   DATA[1350,28] := 263.1056;
   DATA[1350,29] := 11.95847;
   DATA[1350,30] := 1.727378;
   DATA[1350,31] := 1.290893;
   DATA[1350,32] := 0.7353967;
   DATA[1350,33] := 0.3083624;
   DATA[1350,34] := 2.0;
   DATA[1350,35] := 250.3525;
   DATA[1350,36] := 1.681991;
   DATA[1350,37] := 189.0541;
   DATA[1350,38] := 0.000128152;
   DATA[1350,39] := 1.0;
   DATA[1351,1] := 814.22;
   DATA[1351,2] := 1.0;
   DATA[1351,3] := 1.0;
   DATA[1351,4] := 262.5609;
   DATA[1351,5] := 8.462446;
   DATA[1351,6] := 317.9185;
   DATA[1351,8] := 1.0;
   DATA[1351,9] := 1.0;
   DATA[1351,10] := 1.0;
   DATA[1351,11] := 9.47884;
   DATA[1351,12] := 2.225667;
   DATA[1351,13] := 1006.353;
   DATA[1351,14] := 1.0;
   DATA[1351,15] := 1.0;
   DATA[1351,16] := 1.0;
   DATA[1351,17] := 2.0;
   DATA[1351,18] := 1.0;
   DATA[1351,19] := 2.0;
   DATA[1351,20] := 148.808;
   DATA[1351,21] := 154.0374;
   DATA[1351,22] := 1.717489;
   DATA[1351,23] := 791.9893;
   DATA[1351,24] := 2.0;
   DATA[1351,25] := 2.0;
   DATA[1351,26] := 7.87798;
   DATA[1351,27] := 143.0403;
   DATA[1351,28] := 263.1056;
   DATA[1351,29] := 11.95847;
   DATA[1351,30] := 1.726993;
   DATA[1351,31] := 1.291918;
   DATA[1351,32] := 0.7353967;
   DATA[1351,33] := 0.3083624;
   DATA[1351,34] := 2.0;
   DATA[1351,35] := 250.1442;
   DATA[1351,36] := 1.681991;
   DATA[1351,37] := 189.0541;
   DATA[1351,38] := 0.000128152;
   DATA[1351,39] := 1.0;
   DATA[1352,1] := 813.9844;
   DATA[1352,2] := 1.0;
   DATA[1352,3] := 1.0;
   DATA[1352,4] := 262.5609;
   DATA[1352,5] := 8.462446;
   DATA[1352,6] := 317.9185;
   DATA[1352,8] := 1.0;
   DATA[1352,9] := 1.0;
   DATA[1352,10] := 1.0;
   DATA[1352,11] := 9.47884;
   DATA[1352,12] := 2.225667;
   DATA[1352,13] := 1005.752;
   DATA[1352,14] := 1.0;
   DATA[1352,15] := 1.0;
   DATA[1352,16] := 1.0;
   DATA[1352,17] := 2.0;
   DATA[1352,18] := 1.0;
   DATA[1352,19] := 2.0;
   DATA[1352,20] := 148.808;
   DATA[1352,21] := 154.0374;
   DATA[1352,22] := 1.717489;
   DATA[1352,23] := 792.0277;
   DATA[1352,24] := 2.0;
   DATA[1352,25] := 2.0;
   DATA[1352,26] := 7.87798;
   DATA[1352,27] := 142.9121;
   DATA[1352,28] := 263.1056;
   DATA[1352,29] := 11.95847;
   DATA[1352,30] := 1.725455;
   DATA[1352,31] := 1.291918;
   DATA[1352,32] := 0.7353967;
   DATA[1352,33] := 0.3083624;
   DATA[1352,34] := 2.0;
   DATA[1352,35] := 249.984;
   DATA[1352,36] := 1.681991;
   DATA[1352,37] := 188.8458;
   DATA[1352,38] := 0.000128152;
   DATA[1352,39] := 1.0;
   DATA[1353,1] := 814.0237;
   DATA[1353,2] := 1.0;
   DATA[1353,3] := 1.0;
   DATA[1353,4] := 262.5609;
   DATA[1353,5] := 8.462446;
   DATA[1353,6] := 317.9185;
   DATA[1353,8] := 1.0;
   DATA[1353,9] := 1.0;
   DATA[1353,10] := 1.0;
   DATA[1353,11] := 9.47884;
   DATA[1353,12] := 2.225667;
   DATA[1353,13] := 1004.951;
   DATA[1353,14] := 1.0;
   DATA[1353,15] := 1.0;
   DATA[1353,16] := 1.0;
   DATA[1353,17] := 2.0;
   DATA[1353,18] := 1.0;
   DATA[1353,19] := 2.0;
   DATA[1353,20] := 148.808;
   DATA[1353,21] := 154.0374;
   DATA[1353,22] := 1.717489;
   DATA[1353,23] := 791.3356;
   DATA[1353,24] := 2.0;
   DATA[1353,25] := 2.0;
   DATA[1353,26] := 7.87798;
   DATA[1353,27] := 142.9121;
   DATA[1353,28] := 263.1056;
   DATA[1353,29] := 11.95847;
   DATA[1353,30] := 1.724686;
   DATA[1353,31] := 1.291918;
   DATA[1353,32] := 0.7353967;
   DATA[1353,33] := 0.3083624;
   DATA[1353,34] := 2.0;
   DATA[1353,35] := 249.984;
   DATA[1353,36] := 1.681991;
   DATA[1353,37] := 188.8458;
   DATA[1353,38] := 0.000128152;
   DATA[1353,39] := 1.0;
   DATA[1354,1] := 814.22;
   DATA[1354,2] := 1.0;
   DATA[1354,3] := 1.0;
   DATA[1354,4] := 262.5609;
   DATA[1354,5] := 8.462446;
   DATA[1354,6] := 317.9185;
   DATA[1354,8] := 1.0;
   DATA[1354,9] := 1.0;
   DATA[1354,10] := 1.0;
   DATA[1354,11] := 9.430821;
   DATA[1354,12] := 2.225667;
   DATA[1354,13] := 1004.71;
   DATA[1354,14] := 1.0;
   DATA[1354,15] := 1.0;
   DATA[1354,16] := 1.0;
   DATA[1354,17] := 2.0;
   DATA[1354,18] := 1.0;
   DATA[1354,19] := 2.0;
   DATA[1354,20] := 148.808;
   DATA[1354,21] := 154.0374;
   DATA[1354,22] := 1.717105;
   DATA[1354,23] := 791.028;
   DATA[1354,24] := 2.0;
   DATA[1354,25] := 2.0;
   DATA[1354,26] := 7.87798;
   DATA[1354,27] := 142.9121;
   DATA[1354,28] := 263.1056;
   DATA[1354,29] := 11.95847;
   DATA[1354,30] := 1.723532;
   DATA[1354,31] := 1.291918;
   DATA[1354,32] := 0.7353967;
   DATA[1354,33] := 0.3083624;
   DATA[1354,34] := 2.0;
   DATA[1354,35] := 249.984;
   DATA[1354,36] := 1.681991;
   DATA[1354,37] := 188.8458;
   DATA[1354,38] := 0.000128152;
   DATA[1354,39] := 1.0;
   DATA[1355,1] := 814.1415;
   DATA[1355,2] := 1.0;
   DATA[1355,3] := 1.0;
   DATA[1355,4] := 262.5609;
   DATA[1355,5] := 8.462446;
   DATA[1355,6] := 318.021;
   DATA[1355,8] := 1.0;
   DATA[1355,9] := 1.0;
   DATA[1355,10] := 1.0;
   DATA[1355,11] := 9.430821;
   DATA[1355,12] := 2.225667;
   DATA[1355,13] := 1004.31;
   DATA[1355,14] := 1.0;
   DATA[1355,15] := 1.0;
   DATA[1355,16] := 1.0;
   DATA[1355,17] := 2.0;
   DATA[1355,18] := 1.0;
   DATA[1355,19] := 2.0;
   DATA[1355,20] := 148.808;
   DATA[1355,21] := 153.8836;
   DATA[1355,22] := 1.715183;
   DATA[1355,23] := 790.8357;
   DATA[1355,24] := 2.0;
   DATA[1355,25] := 2.0;
   DATA[1355,26] := 7.87798;
   DATA[1355,27] := 142.9121;
   DATA[1355,28] := 263.1056;
   DATA[1355,29] := 11.95847;
   DATA[1355,30] := 1.723532;
   DATA[1355,31] := 1.274241;
   DATA[1355,32] := 0.7353967;
   DATA[1355,33] := 0.3083624;
   DATA[1355,34] := 2.0;
   DATA[1355,35] := 249.984;
   DATA[1355,36] := 1.681991;
   DATA[1355,37] := 188.8458;
   DATA[1355,38] := 0.000128152;
   DATA[1355,39] := 1.0;
   DATA[1356,1] := 813.8275;
   DATA[1356,2] := 1.0;
   DATA[1356,3] := 1.0;
   DATA[1356,4] := 262.5609;
   DATA[1356,5] := 8.462446;
   DATA[1356,6] := 318.021;
   DATA[1356,8] := 1.0;
   DATA[1356,9] := 1.0;
   DATA[1356,10] := 1.0;
   DATA[1356,11] := 9.466035;
   DATA[1356,12] := 2.225667;
   DATA[1356,13] := 1003.949;
   DATA[1356,14] := 1.0;
   DATA[1356,15] := 1.0;
   DATA[1356,16] := 1.0;
   DATA[1356,17] := 2.0;
   DATA[1356,18] := 1.0;
   DATA[1356,19] := 2.0;
   DATA[1356,20] := 148.808;
   DATA[1356,21] := 153.8836;
   DATA[1356,22] := 1.715183;
   DATA[1356,23] := 790.0667;
   DATA[1356,24] := 2.0;
   DATA[1356,25] := 2.0;
   DATA[1356,26] := 7.87798;
   DATA[1356,27] := 142.6045;
   DATA[1356,28] := 263.1056;
   DATA[1356,29] := 11.95847;
   DATA[1356,30] := 1.723532;
   DATA[1356,31] := 1.271039;
   DATA[1356,32] := 0.7353967;
   DATA[1356,33] := 0.3083624;
   DATA[1356,34] := 2.0;
   DATA[1356,35] := 249.984;
   DATA[1356,36] := 1.681991;
   DATA[1356,37] := 188.8458;
   DATA[1356,38] := 0.000128152;
   DATA[1356,39] := 1.0;
   DATA[1357,1] := 813.7489;
   DATA[1357,2] := 1.0;
   DATA[1357,3] := 1.0;
   DATA[1357,4] := 262.5609;
   DATA[1357,5] := 8.462446;
   DATA[1357,6] := 318.021;
   DATA[1357,8] := 1.0;
   DATA[1357,9] := 1.0;
   DATA[1357,10] := 1.0;
   DATA[1357,11] := 9.494846;
   DATA[1357,12] := 2.224898;
   DATA[1357,13] := 1003.509;
   DATA[1357,14] := 1.0;
   DATA[1357,15] := 1.0;
   DATA[1357,16] := 1.0;
   DATA[1357,17] := 2.0;
   DATA[1357,18] := 1.0;
   DATA[1357,19] := 2.0;
   DATA[1357,20] := 148.808;
   DATA[1357,21] := 153.8836;
   DATA[1357,22] := 1.715183;
   DATA[1357,23] := 789.5283;
   DATA[1357,24] := 2.0;
   DATA[1357,25] := 2.0;
   DATA[1357,26] := 7.87798;
   DATA[1357,27] := 142.5788;
   DATA[1357,28] := 263.1056;
   DATA[1357,29] := 11.95847;
   DATA[1357,30] := 1.721866;
   DATA[1357,31] := 1.273601;
   DATA[1357,32] := 0.7353967;
   DATA[1357,33] := 0.3083624;
   DATA[1357,34] := 2.0;
   DATA[1357,35] := 249.984;
   DATA[1357,36] := 1.681991;
   DATA[1357,37] := 188.8458;
   DATA[1357,38] := 0.000128152;
   DATA[1357,39] := 1.0;
   DATA[1358,1] := 813.8275;
   DATA[1358,2] := 1.0;
   DATA[1358,3] := 1.0;
   DATA[1358,4] := 262.5609;
   DATA[1358,5] := 8.464048;
   DATA[1358,6] := 318.021;
   DATA[1358,8] := 1.0;
   DATA[1358,9] := 1.0;
   DATA[1358,10] := 1.0;
   DATA[1358,11] := 9.501248;
   DATA[1358,12] := 2.224898;
   DATA[1358,13] := 1003.349;
   DATA[1358,14] := 1.0;
   DATA[1358,15] := 1.0;
   DATA[1358,16] := 1.0;
   DATA[1358,17] := 2.0;
   DATA[1358,18] := 1.0;
   DATA[1358,19] := 2.0;
   DATA[1358,20] := 148.808;
   DATA[1358,21] := 153.8836;
   DATA[1358,22] := 1.715183;
   DATA[1358,23] := 788.9515;
   DATA[1358,24] := 2.0;
   DATA[1358,25] := 2.0;
   DATA[1358,26] := 7.87798;
   DATA[1358,27] := 142.5788;
   DATA[1358,28] := 263.1056;
   DATA[1358,29] := 11.95847;
   DATA[1358,30] := 1.721866;
   DATA[1358,31] := 1.288331;
   DATA[1358,32] := 0.7353967;
   DATA[1358,33] := 0.3083624;
   DATA[1358,34] := 2.0;
   DATA[1358,35] := 249.984;
   DATA[1358,36] := 1.681991;
   DATA[1358,37] := 188.8458;
   DATA[1358,38] := 0.000128152;
   DATA[1358,39] := 1.0;
   DATA[1359,1] := 814.0237;
   DATA[1359,2] := 1.0;
   DATA[1359,3] := 1.0;
   DATA[1359,4] := 262.5609;
   DATA[1359,5] := 8.46501;
   DATA[1359,6] := 318.021;
   DATA[1359,8] := 1.0;
   DATA[1359,9] := 1.0;
   DATA[1359,10] := 1.0;
   DATA[1359,11] := 9.501248;
   DATA[1359,12] := 2.222592;
   DATA[1359,13] := 1002.948;
   DATA[1359,14] := 1.0;
   DATA[1359,15] := 1.0;
   DATA[1359,16] := 1.0;
   DATA[1359,17] := 2.0;
   DATA[1359,18] := 1.0;
   DATA[1359,19] := 2.0;
   DATA[1359,20] := 148.808;
   DATA[1359,21] := 153.8836;
   DATA[1359,22] := 1.713645;
   DATA[1359,23] := 788.3363;
   DATA[1359,24] := 2.0;
   DATA[1359,25] := 2.0;
   DATA[1359,26] := 7.87798;
   DATA[1359,27] := 142.9121;
   DATA[1359,28] := 263.1056;
   DATA[1359,29] := 12.15073;
   DATA[1359,30] := 1.721866;
   DATA[1359,31] := 1.292686;
   DATA[1359,32] := 0.7353967;
   DATA[1359,33] := 0.3083624;
   DATA[1359,34] := 2.0;
   DATA[1359,35] := 249.984;
   DATA[1359,36] := 1.681991;
   DATA[1359,37] := 188.8458;
   DATA[1359,38] := 0.000128152;
   DATA[1359,39] := 1.0;
   DATA[1360,1] := 813.9059;
   DATA[1360,2] := 1.0;
   DATA[1360,3] := 1.0;
   DATA[1360,4] := 262.5609;
   DATA[1360,5] := 8.46501;
   DATA[1360,6] := 318.021;
   DATA[1360,8] := 1.0;
   DATA[1360,9] := 1.0;
   DATA[1360,10] := 1.0;
   DATA[1360,11] := 9.501248;
   DATA[1360,12] := 2.222592;
   DATA[1360,13] := 1002.908;
   DATA[1360,14] := 1.0;
   DATA[1360,15] := 1.0;
   DATA[1360,16] := 1.0;
   DATA[1360,17] := 2.0;
   DATA[1360,18] := 1.0;
   DATA[1360,19] := 2.0;
   DATA[1360,20] := 148.808;
   DATA[1360,21] := 153.8836;
   DATA[1360,22] := 1.711466;
   DATA[1360,23] := 787.9518;
   DATA[1360,24] := 2.0;
   DATA[1360,25] := 2.0;
   DATA[1360,26] := 7.87798;
   DATA[1360,27] := 142.9121;
   DATA[1360,28] := 263.1056;
   DATA[1360,29] := 12.15073;
   DATA[1360,30] := 1.721866;
   DATA[1360,31] := 1.297938;
   DATA[1360,32] := 0.7353967;
   DATA[1360,33] := 0.3083624;
   DATA[1360,34] := 2.0;
   DATA[1360,35] := 249.984;
   DATA[1360,36] := 1.681991;
   DATA[1360,37] := 188.8458;
   DATA[1360,38] := 0.000128152;
   DATA[1360,39] := 1.0;
   DATA[1361,1] := 813.5527;
   DATA[1361,2] := 1.0;
   DATA[1361,3] := 1.0;
   DATA[1361,4] := 262.5609;
   DATA[1361,5] := 8.46501;
   DATA[1361,6] := 318.021;
   DATA[1361,8] := 1.0;
   DATA[1361,9] := 1.0;
   DATA[1361,10] := 1.0;
   DATA[1361,11] := 9.501248;
   DATA[1361,12] := 2.222592;
   DATA[1361,13] := 1002.267;
   DATA[1361,14] := 1.0;
   DATA[1361,15] := 1.0;
   DATA[1361,16] := 1.0;
   DATA[1361,17] := 2.0;
   DATA[1361,18] := 1.0;
   DATA[1361,19] := 2.0;
   DATA[1361,20] := 148.808;
   DATA[1361,21] := 153.8836;
   DATA[1361,22] := 1.710185;
   DATA[1361,23] := 787.6442;
   DATA[1361,24] := 2.0;
   DATA[1361,25] := 2.0;
   DATA[1361,26] := 7.87798;
   DATA[1361,27] := 142.9121;
   DATA[1361,28] := 263.1056;
   DATA[1361,29] := 12.15073;
   DATA[1361,30] := 1.722507;
   DATA[1361,31] := 1.30114;
   DATA[1361,32] := 0.7353967;
   DATA[1361,33] := 0.3083624;
   DATA[1361,34] := 2.0;
   DATA[1361,35] := 249.984;
   DATA[1361,36] := 1.681991;
   DATA[1361,37] := 188.8458;
   DATA[1361,38] := 0.000128152;
   DATA[1361,39] := 1.0;
   DATA[1362,1] := 813.5919;
   DATA[1362,2] := 1.0;
   DATA[1362,3] := 1.0;
   DATA[1362,4] := 262.5609;
   DATA[1362,5] := 8.46501;
   DATA[1362,6] := 318.021;
   DATA[1362,8] := 1.0;
   DATA[1362,9] := 1.0;
   DATA[1362,10] := 1.0;
   DATA[1362,11] := 9.459633;
   DATA[1362,12] := 2.222592;
   DATA[1362,13] := 1001.947;
   DATA[1362,14] := 1.0;
   DATA[1362,15] := 1.0;
   DATA[1362,16] := 1.0;
   DATA[1362,17] := 2.0;
   DATA[1362,18] := 1.0;
   DATA[1362,19] := 2.0;
   DATA[1362,20] := 148.808;
   DATA[1362,21] := 153.858;
   DATA[1362,22] := 1.710185;
   DATA[1362,23] := 787.2597;
   DATA[1362,24] := 2.0;
   DATA[1362,25] := 2.0;
   DATA[1362,26] := 7.87798;
   DATA[1362,27] := 142.8095;
   DATA[1362,28] := 263.1056;
   DATA[1362,29] := 11.92002;
   DATA[1362,30] := 1.722507;
   DATA[1362,31] := 1.285129;
   DATA[1362,32] := 0.7353967;
   DATA[1362,33] := 0.3083624;
   DATA[1362,34] := 2.0;
   DATA[1362,35] := 249.984;
   DATA[1362,36] := 1.681991;
   DATA[1362,37] := 188.8458;
   DATA[1362,38] := 0.000128152;
   DATA[1362,39] := 1.0;
   DATA[1363,1] := 813.5134;
   DATA[1363,2] := 1.0;
   DATA[1363,3] := 1.0;
   DATA[1363,4] := 262.5609;
   DATA[1363,5] := 8.46501;
   DATA[1363,6] := 318.021;
   DATA[1363,8] := 1.0;
   DATA[1363,9] := 1.0;
   DATA[1363,10] := 1.0;
   DATA[1363,11] := 9.459633;
   DATA[1363,12] := 2.222592;
   DATA[1363,13] := 1001.706;
   DATA[1363,14] := 1.0;
   DATA[1363,16] := 1.0;
   DATA[1363,17] := 2.0;
   DATA[1363,18] := 1.0;
   DATA[1363,19] := 2.0;
   DATA[1363,20] := 148.808;
   DATA[1363,21] := 153.858;
   DATA[1363,22] := 1.70916;
   DATA[1363,23] := 786.8367;
   DATA[1363,24] := 2.0;
   DATA[1363,25] := 2.0;
   DATA[1363,26] := 7.87798;
   DATA[1363,27] := 142.8095;
   DATA[1363,28] := 263.1056;
   DATA[1363,29] := 11.92002;
   DATA[1363,30] := 1.722507;
   DATA[1363,31] := 1.273601;
   DATA[1363,32] := 0.7353967;
   DATA[1363,33] := 0.3083624;
   DATA[1363,34] := 2.0;
   DATA[1363,35] := 249.7757;
   DATA[1363,36] := 1.681991;
   DATA[1363,37] := 188.8458;
   DATA[1363,38] := 0.000128152;
   DATA[1363,39] := 1.0;
   DATA[1364,1] := 813.3564;
   DATA[1364,2] := 1.0;
   DATA[1364,3] := 1.0;
   DATA[1364,4] := 262.5609;
   DATA[1364,5] := 8.46501;
   DATA[1364,6] := 318.021;
   DATA[1364,8] := 1.0;
   DATA[1364,9] := 1.0;
   DATA[1364,10] := 1.0;
   DATA[1364,11] := 9.459633;
   DATA[1364,12] := 2.222592;
   DATA[1364,13] := 1001.506;
   DATA[1364,14] := 1.0;
   DATA[1364,16] := 1.0;
   DATA[1364,17] := 2.0;
   DATA[1364,18] := 1.0;
   DATA[1364,19] := 2.0;
   DATA[1364,20] := 148.808;
   DATA[1364,21] := 153.6529;
   DATA[1364,22] := 1.707109;
   DATA[1364,23] := 785.9139;
   DATA[1364,24] := 2.0;
   DATA[1364,25] := 2.0;
   DATA[1364,26] := 7.87798;
   DATA[1364,27] := 142.8095;
   DATA[1364,28] := 263.1056;
   DATA[1364,29] := 11.92002;
   DATA[1364,30] := 1.722507;
   DATA[1364,31] := 1.263353;
   DATA[1364,32] := 0.7353967;
   DATA[1364,33] := 0.3083624;
   DATA[1364,34] := 2.0;
   DATA[1364,35] := 249.7757;
   DATA[1364,36] := 1.681991;
   DATA[1364,37] := 188.7337;
   DATA[1364,38] := 0.000128152;
   DATA[1364,39] := 1.0;
   DATA[1365,1] := 812.9639;
   DATA[1365,2] := 1.0;
   DATA[1365,3] := 1.0;
   DATA[1365,4] := 262.5609;
   DATA[1365,5] := 8.46501;
   DATA[1365,6] := 318.021;
   DATA[1365,8] := 1.0;
   DATA[1365,9] := 1.0;
   DATA[1365,10] := 1.0;
   DATA[1365,11] := 9.645304;
   DATA[1365,12] := 2.222592;
   DATA[1365,13] := 1000.825;
   DATA[1365,14] := 1.0;
   DATA[1365,16] := 1.0;
   DATA[1365,17] := 2.0;
   DATA[1365,18] := 1.0;
   DATA[1365,19] := 2.0;
   DATA[1365,20] := 148.808;
   DATA[1365,21] := 153.6529;
   DATA[1365,22] := 1.705571;
   DATA[1365,23] := 785.7601;
   DATA[1365,24] := 2.0;
   DATA[1365,25] := 2.0;
   DATA[1365,26] := 7.87798;
   DATA[1365,27] := 142.8095;
   DATA[1365,28] := 263.1056;
   DATA[1365,29] := 11.92002;
   DATA[1365,30] := 1.722507;
   DATA[1365,31] := 1.262457;
   DATA[1365,32] := 0.7353967;
   DATA[1365,33] := 0.3083624;
   DATA[1365,34] := 2.0;
   DATA[1365,35] := 249.7757;
   DATA[1365,36] := 1.681991;
   DATA[1365,37] := 188.6535;
   DATA[1365,38] := 0.000128152;
   DATA[1365,39] := 1.0;
   DATA[1366,1] := 813.1602;
   DATA[1366,2] := 1.0;
   DATA[1366,3] := 1.0;
   DATA[1366,4] := 262.5609;
   DATA[1366,5] := 8.46501;
   DATA[1366,6] := 318.021;
   DATA[1366,8] := 1.0;
   DATA[1366,9] := 1.0;
   DATA[1366,10] := 1.0;
   DATA[1366,11] := 10.06787;
   DATA[1366,12] := 2.222592;
   DATA[1366,13] := 1000.344;
   DATA[1366,14] := 1.0;
   DATA[1366,16] := 1.0;
   DATA[1366,17] := 2.0;
   DATA[1366,18] := 1.0;
   DATA[1366,19] := 2.0;
   DATA[1366,20] := 148.808;
   DATA[1366,21] := 153.6529;
   DATA[1366,22] := 1.705571;
   DATA[1366,23] := 785.6832;
   DATA[1366,24] := 2.0;
   DATA[1366,25] := 2.0;
   DATA[1366,26] := 7.87798;
   DATA[1366,27] := 142.8095;
   DATA[1366,28] := 263.1056;
   DATA[1366,29] := 11.92002;
   DATA[1366,30] := 1.722507;
   DATA[1366,31] := 1.26758;
   DATA[1366,32] := 0.7353967;
   DATA[1366,33] := 0.3083624;
   DATA[1366,34] := 2.0;
   DATA[1366,35] := 249.7757;
   DATA[1366,36] := 1.681991;
   DATA[1366,37] := 188.6535;
   DATA[1366,38] := 0.000128152;
   DATA[1366,39] := 1.0;
   DATA[1367,1] := 813.1994;
   DATA[1367,2] := 1.0;
   DATA[1367,3] := 1.0;
   DATA[1367,4] := 262.5609;
   DATA[1367,5] := 8.46501;
   DATA[1367,6] := 318.1748;
   DATA[1367,8] := 1.0;
   DATA[1367,9] := 1.0;
   DATA[1367,10] := 1.0;
   DATA[1367,11] := 10.58326;
   DATA[1367,12] := 2.234635;
   DATA[1367,13] := 1000.344;
   DATA[1367,14] := 1.0;
   DATA[1367,16] := 1.0;
   DATA[1367,17] := 2.0;
   DATA[1367,18] := 1.0;
   DATA[1367,19] := 2.0;
   DATA[1367,20] := 148.808;
   DATA[1367,21] := 153.7554;
   DATA[1367,22] := 1.705059;
   DATA[1367,23] := 785.2602;
   DATA[1367,24] := 2.0;
   DATA[1367,25] := 2.0;
   DATA[1367,26] := 7.87798;
   DATA[1367,27] := 142.8095;
   DATA[1367,28] := 263.1056;
   DATA[1367,29] := 11.92002;
   DATA[1367,30] := 1.722507;
   DATA[1367,31] := 1.266299;
   DATA[1367,32] := 0.7368051;
   DATA[1367,33] := 0.3083624;
   DATA[1367,34] := 2.0;
   DATA[1367,35] := 249.5995;
   DATA[1367,36] := 1.681991;
   DATA[1367,37] := 188.4613;
   DATA[1367,38] := 0.000128152;
   DATA[1367,39] := 1.0;
   DATA[1368,1] := 812.6498;
   DATA[1368,2] := 1.0;
   DATA[1368,3] := 1.0;
   DATA[1368,4] := 262.5609;
   DATA[1368,5] := 8.46501;
   DATA[1368,6] := 318.1748;
   DATA[1368,8] := 1.0;
   DATA[1368,9] := 1.0;
   DATA[1368,10] := 1.0;
   DATA[1368,11] := 11.10186;
   DATA[1368,12] := 2.243731;
   DATA[1368,13] := 1000.024;
   DATA[1368,14] := 1.0;
   DATA[1368,16] := 1.0;
   DATA[1368,17] := 2.0;
   DATA[1368,18] := 1.0;
   DATA[1368,19] := 2.0;
   DATA[1368,20] := 148.808;
   DATA[1368,21] := 153.8067;
   DATA[1368,22] := 1.703905;
   DATA[1368,23] := 784.9141;
   DATA[1368,24] := 2.0;
   DATA[1368,25] := 2.0;
   DATA[1368,26] := 7.87798;
   DATA[1368,27] := 142.8095;
   DATA[1368,28] := 263.1056;
   DATA[1368,29] := 12.03538;
   DATA[1368,30] := 1.722507;
   DATA[1368,31] := 1.266299;
   DATA[1368,32] := 0.7377012;
   DATA[1368,33] := 0.3083624;
   DATA[1368,34] := 2.0;
   DATA[1368,35] := 249.5834;
   DATA[1368,36] := 1.681991;
   DATA[1368,37] := 188.4613;
   DATA[1368,38] := 0.000128152;
   DATA[1368,39] := 1.0;
   DATA[1369,1] := 813.0424;
   DATA[1369,2] := 1.0;
   DATA[1369,3] := 1.0;
   DATA[1369,4] := 262.5609;
   DATA[1369,5] := 8.46501;
   DATA[1369,6] := 318.1748;
   DATA[1369,8] := 1.0;
   DATA[1369,9] := 1.0;
   DATA[1369,10] := 1.0;
   DATA[1369,11] := 11.62366;
   DATA[1369,12] := 2.26141;
   DATA[1369,13] := 999.7437;
   DATA[1369,14] := 1.0;
   DATA[1369,16] := 1.0;
   DATA[1369,17] := 2.0;
   DATA[1369,18] := 1.0;
   DATA[1369,19] := 2.0;
   DATA[1369,20] := 148.808;
   DATA[1369,21] := 153.8067;
   DATA[1369,22] := 1.703905;
   DATA[1369,23] := 784.4142;
   DATA[1369,24] := 2.0;
   DATA[1369,25] := 2.0;
   DATA[1369,26] := 7.87798;
   DATA[1369,27] := 142.8095;
   DATA[1369,28] := 263.1056;
   DATA[1369,29] := 12.03538;
   DATA[1369,30] := 1.721866;
   DATA[1369,31] := 1.254259;
   DATA[1369,32] := 0.7357808;
   DATA[1369,33] := 0.3083624;
   DATA[1369,34] := 2.0;
   DATA[1369,35] := 249.5834;
   DATA[1369,36] := 1.681991;
   DATA[1369,37] := 188.4613;
   DATA[1369,38] := 0.000128152;
   DATA[1369,39] := 1.0;
   DATA[1370,1] := 813.1209;
   DATA[1370,2] := 1.0;
   DATA[1370,3] := 1.0;
   DATA[1370,4] := 262.5609;
   DATA[1370,5] := 8.46501;
   DATA[1370,6] := 318.1748;
   DATA[1370,8] := 1.0;
   DATA[1370,9] := 1.0;
   DATA[1370,10] := 1.0;
   DATA[1370,11] := 12.14546;
   DATA[1370,12] := 2.278192;
   DATA[1370,13] := 999.223;
   DATA[1370,14] := 1.0;
   DATA[1370,15] := 2.0;
   DATA[1370,16] := 1.0;
   DATA[1370,17] := 2.0;
   DATA[1370,18] := 1.0;
   DATA[1370,19] := 2.0;
   DATA[1370,20] := 148.808;
   DATA[1370,21] := 153.8067;
   DATA[1370,22] := 1.703905;
   DATA[1370,23] := 784.7219;
   DATA[1370,24] := 2.0;
   DATA[1370,25] := 2.0;
   DATA[1370,26] := 7.87798;
   DATA[1370,27] := 142.8095;
   DATA[1370,28] := 263.1056;
   DATA[1370,29] := 12.03538;
   DATA[1370,30] := 1.721866;
   DATA[1370,31] := 1.2549;
   DATA[1370,32] := 0.7355248;
   DATA[1370,33] := 0.3083624;
   DATA[1370,34] := 2.0;
   DATA[1370,35] := 249.5834;
   DATA[1370,36] := 1.681991;
   DATA[1370,37] := 188.4613;
   DATA[1370,38] := 0.000128152;
   DATA[1370,39] := 1.0;
   DATA[1371,1] := 812.9639;
   DATA[1371,2] := 1.0;
   DATA[1371,3] := 1.0;
   DATA[1371,4] := 262.5609;
   DATA[1371,5] := 8.46501;
   DATA[1371,6] := 318.1748;
   DATA[1371,8] := 1.0;
   DATA[1371,9] := 1.0;
   DATA[1371,10] := 1.0;
   DATA[1371,11] := 12.66726;
   DATA[1371,12] := 2.298049;
   DATA[1371,13] := 998.8625;
   DATA[1371,14] := 1.0;
   DATA[1371,15] := 2.0;
   DATA[1371,16] := 1.0;
   DATA[1371,18] := 1.0;
   DATA[1371,19] := 2.0;
   DATA[1371,20] := 148.808;
   DATA[1371,21] := 153.8067;
   DATA[1371,22] := 1.7057;
   DATA[1371,23] := 783.9913;
   DATA[1371,24] := 2.0;
   DATA[1371,25] := 2.0;
   DATA[1371,26] := 7.87798;
   DATA[1371,27] := 142.8608;
   DATA[1371,28] := 263.1056;
   DATA[1371,29] := 12.03538;
   DATA[1371,30] := 1.721866;
   DATA[1371,31] := 1.275906;
   DATA[1371,32] := 0.7347566;
   DATA[1371,33] := 0.3083624;
   DATA[1371,34] := 2.0;
   DATA[1371,35] := 249.7116;
   DATA[1371,36] := 1.681991;
   DATA[1371,37] := 188.6375;
   DATA[1371,38] := 0.000128152;
   DATA[1371,39] := 1.0;
   DATA[1372,1] := 812.7283;
   DATA[1372,2] := 1.0;
   DATA[1372,3] := 1.0;
   DATA[1372,4] := 262.5609;
   DATA[1372,5] := 8.46501;
   DATA[1372,6] := 318.1748;
   DATA[1372,8] := 1.0;
   DATA[1372,9] := 1.0;
   DATA[1372,10] := 1.0;
   DATA[1372,11] := 13.12184;
   DATA[1372,12] := 2.312013;
   DATA[1372,13] := 998.4219;
   DATA[1372,14] := 1.0;
   DATA[1372,15] := 2.0;
   DATA[1372,16] := 1.0;
   DATA[1372,18] := 1.0;
   DATA[1372,19] := 2.0;
   DATA[1372,20] := 148.808;
   DATA[1372,21] := 153.8067;
   DATA[1372,22] := 1.7098;
   DATA[1372,23] := 783.9144;
   DATA[1372,24] := 2.0;
   DATA[1372,25] := 2.0;
   DATA[1372,26] := 7.87798;
   DATA[1372,27] := 142.8608;
   DATA[1372,28] := 263.1056;
   DATA[1372,29] := 12.03538;
   DATA[1372,30] := 1.721866;
   DATA[1372,31] := 1.293711;
   DATA[1372,32] := 0.7347566;
   DATA[1372,33] := 0.3083624;
   DATA[1372,34] := 2.0;
   DATA[1372,35] := 249.8718;
   DATA[1372,36] := 1.681991;
   DATA[1372,37] := 188.7977;
   DATA[1372,38] := 0.000128152;
   DATA[1372,39] := 1.0;
   DATA[1373,1] := 812.9639;
   DATA[1373,2] := 1.0;
   DATA[1373,3] := 1.0;
   DATA[1373,4] := 262.5609;
   DATA[1373,5] := 8.46501;
   DATA[1373,6] := 318.1748;
   DATA[1373,8] := 1.0;
   DATA[1373,9] := 1.0;
   DATA[1373,10] := 1.0;
   DATA[1373,11] := 13.2755;
   DATA[1373,12] := 2.321237;
   DATA[1373,13] := 997.8211;
   DATA[1373,14] := 1.0;
   DATA[1373,15] := 2.0;
   DATA[1373,16] := 1.0;
   DATA[1373,18] := 1.0;
   DATA[1373,19] := 2.0;
   DATA[1373,20] := 148.808;
   DATA[1373,21] := 153.8067;
   DATA[1373,22] := 1.710313;
   DATA[1373,23] := 783.6068;
   DATA[1373,24] := 2.0;
   DATA[1373,25] := 2.0;
   DATA[1373,26] := 7.87798;
   DATA[1373,27] := 142.8608;
   DATA[1373,28] := 263.1056;
   DATA[1373,29] := 12.03538;
   DATA[1373,30] := 1.722123;
   DATA[1373,31] := 1.310619;
   DATA[1373,32] := 0.7347566;
   DATA[1373,33] := 0.3083624;
   DATA[1373,34] := 2.0;
   DATA[1373,35] := 250.0;
   DATA[1373,36] := 1.681991;
   DATA[1373,37] := 188.8458;
   DATA[1373,38] := 0.000128152;
   DATA[1373,39] := 1.0;
   DATA[1374,1] := 813.0031;
   DATA[1374,2] := 1.0;
   DATA[1374,3] := 1.0;
   DATA[1374,4] := 262.5609;
   DATA[1374,5] := 8.46501;
   DATA[1374,6] := 318.1748;
   DATA[1374,8] := 1.0;
   DATA[1374,9] := 1.0;
   DATA[1374,10] := 1.0;
   DATA[1374,11] := 13.37794;
   DATA[1374,12] := 2.327003;
   DATA[1374,13] := 997.5007;
   DATA[1374,14] := 1.0;
   DATA[1374,15] := 2.0;
   DATA[1374,16] := 1.0;
   DATA[1374,18] := 1.0;
   DATA[1374,19] := 2.0;
   DATA[1374,20] := 148.808;
   DATA[1374,21] := 153.8067;
   DATA[1374,22] := 1.712235;
   DATA[1374,23] := 783.2607;
   DATA[1374,24] := 2.0;
   DATA[1374,25] := 2.0;
   DATA[1374,26] := 7.87798;
   DATA[1374,27] := 142.8608;
   DATA[1374,28] := 263.1056;
   DATA[1374,29] := 12.03538;
   DATA[1374,30] := 1.72443;
   DATA[1374,31] := 1.309466;
   DATA[1374,32] := 0.7351407;
   DATA[1374,33] := 0.3083624;
   DATA[1374,34] := 2.0;
   DATA[1374,35] := 250.0961;
   DATA[1374,36] := 1.681991;
   DATA[1374,37] := 188.8458;
   DATA[1374,38] := 0.000128152;
   DATA[1374,39] := 1.0;
   DATA[1375,1] := 812.7283;
   DATA[1375,2] := 1.0;
   DATA[1375,3] := 1.0;
   DATA[1375,4] := 262.5609;
   DATA[1375,5] := 8.46501;
   DATA[1375,6] := 318.1748;
   DATA[1375,8] := 1.0;
   DATA[1375,9] := 1.0;
   DATA[1375,10] := 1.0;
   DATA[1375,11] := 13.62763;
   DATA[1375,12] := 2.328668;
   DATA[1375,13] := 996.9399;
   DATA[1375,14] := 1.0;
   DATA[1375,15] := 2.0;
   DATA[1375,16] := 1.0;
   DATA[1375,18] := 1.0;
   DATA[1375,19] := 2.0;
   DATA[1375,20] := 148.808;
   DATA[1375,21] := 153.8067;
   DATA[1375,22] := 1.714029;
   DATA[1375,23] := 783.1453;
   DATA[1375,24] := 2.0;
   DATA[1375,25] := 2.0;
   DATA[1375,26] := 7.87798;
   DATA[1375,27] := 142.8608;
   DATA[1375,28] := 263.1056;
   DATA[1375,29] := 12.03538;
   DATA[1375,30] := 1.72443;
   DATA[1375,31] := 1.29243;
   DATA[1375,32] := 0.7359089;
   DATA[1375,33] := 0.3083624;
   DATA[1375,34] := 2.0;
   DATA[1375,35] := 250.1602;
   DATA[1375,36] := 1.681991;
   DATA[1375,37] := 189.022;
   DATA[1375,38] := 0.000128152;
   DATA[1375,39] := 1.0;
   DATA[1376,1] := 812.9639;
   DATA[1376,2] := 1.0;
   DATA[1376,3] := 1.0;
   DATA[1376,4] := 262.5609;
   DATA[1376,5] := 8.46501;
   DATA[1376,6] := 318.1748;
   DATA[1376,8] := 1.0;
   DATA[1376,9] := 1.0;
   DATA[1376,10] := 1.0;
   DATA[1376,11] := 13.92535;
   DATA[1376,12] := 2.328668;
   DATA[1376,13] := 996.7396;
   DATA[1376,14] := 1.0;
   DATA[1376,15] := 2.0;
   DATA[1376,16] := 1.0;
   DATA[1376,18] := 1.0;
   DATA[1376,19] := 2.0;
   DATA[1376,20] := 148.808;
   DATA[1376,21] := 153.8067;
   DATA[1376,22] := 1.714798;
   DATA[1376,23] := 782.607;
   DATA[1376,24] := 2.0;
   DATA[1376,25] := 2.0;
   DATA[1376,26] := 7.87798;
   DATA[1376,27] := 142.8608;
   DATA[1376,28] := 263.1056;
   DATA[1376,29] := 12.03538;
   DATA[1376,30] := 1.72443;
   DATA[1376,31] := 1.291277;
   DATA[1376,32] := 0.7359089;
   DATA[1376,33] := 0.3083624;
   DATA[1376,34] := 2.0;
   DATA[1376,35] := 250.1602;
   DATA[1376,36] := 1.681991;
   DATA[1376,37] := 189.022;
   DATA[1376,38] := 0.000128152;
   DATA[1376,39] := 1.0;
   DATA[1377,1] := 813.0424;
   DATA[1377,2] := 1.0;
   DATA[1377,3] := 1.0;
   DATA[1377,4] := 262.5609;
   DATA[1377,5] := 8.46501;
   DATA[1377,6] := 318.1748;
   DATA[1377,8] := 1.0;
   DATA[1377,9] := 1.0;
   DATA[1377,10] := 1.0;
   DATA[1377,11] := 14.40233;
   DATA[1377,12] := 2.328668;
   DATA[1377,13] := 996.0988;
   DATA[1377,14] := 1.0;
   DATA[1377,15] := 2.0;
   DATA[1377,16] := 1.0;
   DATA[1377,18] := 1.0;
   DATA[1377,19] := 2.0;
   DATA[1377,20] := 148.808;
   DATA[1377,21] := 153.8067;
   DATA[1377,22] := 1.715824;
   DATA[1377,23] := 782.1841;
   DATA[1377,24] := 2.0;
   DATA[1377,25] := 2.0;
   DATA[1377,26] := 7.87798;
   DATA[1377,27] := 142.8608;
   DATA[1377,28] := 263.1056;
   DATA[1377,29] := 12.03538;
   DATA[1377,30] := 1.724173;
   DATA[1377,31] := 1.281286;
   DATA[1377,32] := 0.7359089;
   DATA[1377,33] := 0.3083624;
   DATA[1377,34] := 2.0;
   DATA[1377,35] := 250.1923;
   DATA[1377,36] := 1.681991;
   DATA[1377,37] := 189.1823;
   DATA[1377,38] := 0.000128152;
   DATA[1377,39] := 1.0;
   DATA[1378,1] := 813.5527;
   DATA[1378,2] := 1.0;
   DATA[1378,3] := 1.0;
   DATA[1378,4] := 262.5609;
   DATA[1378,5] := 8.46501;
   DATA[1378,6] := 318.1748;
   DATA[1378,8] := 1.0;
   DATA[1378,9] := 1.0;
   DATA[1378,10] := 1.0;
   DATA[1378,11] := 14.91453;
   DATA[1378,12] := 2.323672;
   DATA[1378,13] := 995.2977;
   DATA[1378,14] := 1.0;
   DATA[1378,15] := 2.0;
   DATA[1378,16] := 1.0;
   DATA[1378,17] := 1.0;
   DATA[1378,18] := 1.0;
   DATA[1378,19] := 2.0;
   DATA[1378,20] := 148.808;
   DATA[1378,21] := 153.7554;
   DATA[1378,22] := 1.715824;
   DATA[1378,23] := 782.0687;
   DATA[1378,24] := 2.0;
   DATA[1378,25] := 2.0;
   DATA[1378,26] := 7.87798;
   DATA[1378,27] := 142.8608;
   DATA[1378,28] := 263.1056;
   DATA[1378,29] := 12.03538;
   DATA[1378,30] := 1.723148;
   DATA[1378,31] := 1.281286;
   DATA[1378,32] := 0.7359089;
   DATA[1378,33] := 0.3083624;
   DATA[1378,34] := 2.0;
   DATA[1378,35] := 250.1923;
   DATA[1378,36] := 1.762086;
   DATA[1378,37] := 189.1823;
   DATA[1378,38] := 0.000128152;
   DATA[1378,39] := 1.0;
   DATA[1379,1] := 813.5527;
   DATA[1379,2] := 1.0;
   DATA[1379,3] := 1.0;
   DATA[1379,4] := 262.5609;
   DATA[1379,5] := 8.46501;
   DATA[1379,6] := 318.1748;
   DATA[1379,8] := 1.0;
   DATA[1379,9] := 1.0;
   DATA[1379,10] := 1.0;
   DATA[1379,11] := 15.43633;
   DATA[1379,12] := 2.313423;
   DATA[1379,13] := 994.8972;
   DATA[1379,14] := 1.0;
   DATA[1379,15] := 2.0;
   DATA[1379,16] := 1.0;
   DATA[1379,17] := 1.0;
   DATA[1379,18] := 1.0;
   DATA[1379,19] := 2.0;
   DATA[1379,20] := 148.808;
   DATA[1379,21] := 153.7554;
   DATA[1379,22] := 1.715824;
   DATA[1379,23] := 781.838;
   DATA[1379,24] := 2.0;
   DATA[1379,25] := 2.0;
   DATA[1379,26] := 7.87798;
   DATA[1379,27] := 142.8608;
   DATA[1379,28] := 263.1056;
   DATA[1379,29] := 12.26609;
   DATA[1379,30] := 1.723148;
   DATA[1379,31] := 1.27232;
   DATA[1379,32] := 0.7355248;
   DATA[1379,33] := 0.3083624;
   DATA[1379,34] := 2.0;
   DATA[1379,35] := 250.1923;
   DATA[1379,36] := 1.762086;
   DATA[1379,37] := 189.1823;
   DATA[1379,38] := 0.000128152;
   DATA[1379,39] := 1.0;
   DATA[1380,1] := 813.3171;
   DATA[1380,2] := 1.0;
   DATA[1380,3] := 1.0;
   DATA[1380,4] := 262.5609;
   DATA[1380,5] := 8.46501;
   DATA[1380,6] := 318.1748;
   DATA[1380,8] := 1.0;
   DATA[1380,9] := 1.0;
   DATA[1380,10] := 1.0;
   DATA[1380,11] := 16.03176;
   DATA[1380,12] := 2.302661;
   DATA[1380,13] := 994.1362;
   DATA[1380,14] := 1.0;
   DATA[1380,15] := 2.0;
   DATA[1380,16] := 1.0;
   DATA[1380,17] := 1.0;
   DATA[1380,18] := 1.0;
   DATA[1380,19] := 2.0;
   DATA[1380,20] := 148.808;
   DATA[1380,21] := 153.6273;
   DATA[1380,22] := 1.715183;
   DATA[1380,23] := 781.4919;
   DATA[1380,24] := 2.0;
   DATA[1380,25] := 2.0;
   DATA[1380,26] := 7.87798;
   DATA[1380,27] := 142.989;
   DATA[1380,28] := 263.1056;
   DATA[1380,29] := 12.26609;
   DATA[1380,30] := 1.723148;
   DATA[1380,31] := 1.271679;
   DATA[1380,32] := 0.7355248;
   DATA[1380,33] := 0.3083624;
   DATA[1380,34] := 2.0;
   DATA[1380,35] := 250.1923;
   DATA[1380,36] := 1.762086;
   DATA[1380,37] := 189.006;
   DATA[1380,38] := 0.000128152;
   DATA[1380,39] := 1.0;
   DATA[1381,1] := 813.1602;
   DATA[1381,2] := 1.0;
   DATA[1381,3] := 1.0;
   DATA[1381,4] := 262.5609;
   DATA[1381,5] := 8.46501;
   DATA[1381,6] := 318.1748;
   DATA[1381,8] := 1.0;
   DATA[1381,9] := 1.0;
   DATA[1381,10] := 1.0;
   DATA[1381,11] := 16.80645;
   DATA[1381,12] := 2.284085;
   DATA[1381,13] := 993.5353;
   DATA[1381,14] := 1.0;
   DATA[1381,15] := 2.0;
   DATA[1381,16] := 1.0;
   DATA[1381,17] := 1.0;
   DATA[1381,18] := 1.0;
   DATA[1381,19] := 2.0;
   DATA[1381,20] := 148.808;
   DATA[1381,21] := 153.6273;
   DATA[1381,22] := 1.714798;
   DATA[1381,23] := 781.1459;
   DATA[1381,24] := 2.0;
   DATA[1381,25] := 2.0;
   DATA[1381,26] := 7.87798;
   DATA[1381,27] := 142.989;
   DATA[1381,28] := 263.1056;
   DATA[1381,29] := 12.26609;
   DATA[1381,30] := 1.723148;
   DATA[1381,31] := 1.279749;
   DATA[1381,32] := 0.7355248;
   DATA[1381,33] := 0.3083624;
   DATA[1381,34] := 2.0;
   DATA[1381,35] := 250.1923;
   DATA[1381,36] := 1.649953;
   DATA[1381,37] := 188.9259;
   DATA[1381,38] := 0.000128152;
   DATA[1381,39] := 1.0;
   DATA[1382,1] := 813.5919;
   DATA[1382,2] := 1.0;
   DATA[1382,3] := 1.0;
   DATA[1382,4] := 262.5609;
   DATA[1382,5] := 8.46501;
   DATA[1382,6] := 318.1748;
   DATA[1382,8] := 1.0;
   DATA[1382,9] := 1.0;
   DATA[1382,10] := 1.0;
   DATA[1382,11] := 17.50752;
   DATA[1382,12] := 2.267175;
   DATA[1382,13] := 993.0547;
   DATA[1382,14] := 1.0;
   DATA[1382,15] := 2.0;
   DATA[1382,16] := 1.0;
   DATA[1382,17] := 1.0;
   DATA[1382,18] := 1.0;
   DATA[1382,19] := 2.0;
   DATA[1382,20] := 148.808;
   DATA[1382,21] := 153.6273;
   DATA[1382,22] := 1.714798;
   DATA[1382,23] := 780.9536;
   DATA[1382,24] := 2.0;
   DATA[1382,25] := 2.0;
   DATA[1382,26] := 7.87798;
   DATA[1382,27] := 142.989;
   DATA[1382,28] := 263.1056;
   DATA[1382,29] := 12.26609;
   DATA[1382,30] := 1.724173;
   DATA[1382,31] := 1.291405;
   DATA[1382,32] := 0.7355248;
   DATA[1382,33] := 0.3083624;
   DATA[1382,34] := 2.0;
   DATA[1382,35] := 250.1923;
   DATA[1382,36] := 1.649953;
   DATA[1382,37] := 188.9259;
   DATA[1382,38] := 0.000128152;
   DATA[1382,39] := 1.0;
   DATA[1383,1] := 813.3171;
   DATA[1383,2] := 1.0;
   DATA[1383,3] := 1.0;
   DATA[1383,4] := 262.5609;
   DATA[1383,5] := 8.46501;
   DATA[1383,6] := 318.1748;
   DATA[1383,8] := 1.0;
   DATA[1383,9] := 1.0;
   DATA[1383,10] := 1.0;
   DATA[1383,11] := 18.05493;
   DATA[1383,12] := 2.247318;
   DATA[1383,13] := 992.8544;
   DATA[1383,14] := 1.0;
   DATA[1383,15] := 2.0;
   DATA[1383,16] := 1.0;
   DATA[1383,17] := 1.0;
   DATA[1383,18] := 1.0;
   DATA[1383,19] := 2.0;
   DATA[1383,20] := 148.808;
   DATA[1383,21] := 153.6273;
   DATA[1383,22] := 1.712107;
   DATA[1383,23] := 780.9536;
   DATA[1383,24] := 2.0;
   DATA[1383,25] := 2.0;
   DATA[1383,26] := 7.87798;
   DATA[1383,27] := 142.989;
   DATA[1383,28] := 263.1056;
   DATA[1383,29] := 12.11228;
   DATA[1383,30] := 1.724173;
   DATA[1383,31] := 1.291405;
   DATA[1383,32] := 0.7355248;
   DATA[1383,33] := 0.3083624;
   DATA[1383,34] := 2.0;
   DATA[1383,35] := 249.8398;
   DATA[1383,36] := 1.601897;
   DATA[1383,37] := 188.9259;
   DATA[1383,38] := 0.000128152;
   DATA[1383,39] := 1.0;
   DATA[1384,1] := 813.5527;
   DATA[1384,2] := 1.0;
   DATA[1384,3] := 1.0;
   DATA[1384,4] := 262.5609;
   DATA[1384,5] := 8.46501;
   DATA[1384,6] := 318.1748;
   DATA[1384,8] := 1.0;
   DATA[1384,9] := 1.0;
   DATA[1384,10] := 1.0;
   DATA[1384,11] := 18.57994;
   DATA[1384,12] := 2.234378;
   DATA[1384,13] := 992.4138;
   DATA[1384,14] := 1.0;
   DATA[1384,15] := 2.0;
   DATA[1384,16] := 1.0;
   DATA[1384,17] := 1.0;
   DATA[1384,18] := 1.0;
   DATA[1384,19] := 2.0;
   DATA[1384,20] := 148.808;
   DATA[1384,21] := 153.6273;
   DATA[1384,22] := 1.712107;
   DATA[1384,23] := 780.4153;
   DATA[1384,24] := 2.0;
   DATA[1384,25] := 2.0;
   DATA[1384,26] := 7.87798;
   DATA[1384,27] := 142.989;
   DATA[1384,28] := 263.1056;
   DATA[1384,29] := 12.11228;
   DATA[1384,30] := 1.724173;
   DATA[1384,31] := 1.291405;
   DATA[1384,32] := 0.7355248;
   DATA[1384,33] := 0.3083624;
   DATA[1384,34] := 2.0;
   DATA[1384,35] := 249.8398;
   DATA[1384,36] := 1.601897;
   DATA[1384,37] := 188.6535;
   DATA[1384,38] := 0.000128152;
   DATA[1384,39] := 1.0;
   DATA[1385,1] := 813.4349;
   DATA[1385,2] := 1.0;
   DATA[1385,3] := 1.0;
   DATA[1385,4] := 262.5609;
   DATA[1385,5] := 8.46501;
   DATA[1385,6] := 318.1236;
   DATA[1385,8] := 1.0;
   DATA[1385,9] := 1.0;
   DATA[1385,10] := 1.0;
   DATA[1385,11] := 19.09853;
   DATA[1385,12] := 2.224258;
   DATA[1385,13] := 992.2936;
   DATA[1385,14] := 1.0;
   DATA[1385,15] := 2.0;
   DATA[1385,16] := 1.0;
   DATA[1385,17] := 1.0;
   DATA[1385,18] := 1.0;
   DATA[1385,19] := 2.0;
   DATA[1385,20] := 148.808;
   DATA[1385,21] := 153.4991;
   DATA[1385,22] := 1.712107;
   DATA[1385,23] := 780.223;
   DATA[1385,24] := 2.0;
   DATA[1385,25] := 2.0;
   DATA[1385,26] := 7.87798;
   DATA[1385,27] := 142.989;
   DATA[1385,28] := 263.1056;
   DATA[1385,29] := 12.11228;
   DATA[1385,30] := 1.724173;
   DATA[1385,31] := 1.285385;
   DATA[1385,32] := 0.7355248;
   DATA[1385,33] := 0.3083624;
   DATA[1385,34] := 2.0;
   DATA[1385,35] := 249.8398;
   DATA[1385,36] := 1.601897;
   DATA[1385,37] := 188.6215;
   DATA[1385,38] := 0.000128152;
   DATA[1385,39] := 1.0;
   DATA[1386,1] := 813.6312;
   DATA[1386,2] := 1.0;
   DATA[1386,3] := 1.0;
   DATA[1386,4] := 262.5609;
   DATA[1386,5] := 8.46501;
   DATA[1386,6] := 318.1236;
   DATA[1386,8] := 1.0;
   DATA[1386,9] := 1.0;
   DATA[1386,10] := 1.0;
   DATA[1386,11] := 19.5403;
   DATA[1386,12] := 2.222336;
   DATA[1386,13] := 991.7329;
   DATA[1386,14] := 1.0;
   DATA[1386,15] := 2.0;
   DATA[1386,16] := 1.0;
   DATA[1386,17] := 1.0;
   DATA[1386,18] := 1.0;
   DATA[1386,19] := 2.0;
   DATA[1386,20] := 148.808;
   DATA[1386,21] := 153.4991;
   DATA[1386,22] := 1.712107;
   DATA[1386,23] := 780.0692;
   DATA[1386,24] := 2.0;
   DATA[1386,25] := 2.0;
   DATA[1386,26] := 7.87798;
   DATA[1386,27] := 142.8095;
   DATA[1386,28] := 263.1056;
   DATA[1386,29] := 12.11228;
   DATA[1386,30] := 1.721225;
   DATA[1386,31] := 1.281542;
   DATA[1386,32] := 0.7355248;
   DATA[1386,33] := 0.3083624;
   DATA[1386,34] := 2.0;
   DATA[1386,35] := 249.5995;
   DATA[1386,36] := 1.601897;
   DATA[1386,37] := 188.5734;
   DATA[1386,38] := 0.000128152;
   DATA[1386,39] := 1.0;
   DATA[1387,1] := 813.5527;
   DATA[1387,2] := 1.0;
   DATA[1387,3] := 1.0;
   DATA[1387,4] := 262.5609;
   DATA[1387,5] := 8.46501;
   DATA[1387,6] := 318.1236;
   DATA[1387,8] := 1.0;
   DATA[1387,9] := 1.0;
   DATA[1387,10] := 1.0;
   DATA[1387,11] := 19.65555;
   DATA[1387,12] := 2.220542;
   DATA[1387,13] := 991.3324;
   DATA[1387,14] := 1.0;
   DATA[1387,15] := 2.0;
   DATA[1387,16] := 1.0;
   DATA[1387,17] := 1.0;
   DATA[1387,18] := 1.0;
   DATA[1387,19] := 2.0;
   DATA[1387,20] := 148.808;
   DATA[1387,21] := 153.4991;
   DATA[1387,22] := 1.712107;
   DATA[1387,23] := 779.877;
   DATA[1387,24] := 2.0;
   DATA[1387,25] := 2.0;
   DATA[1387,26] := 7.87798;
   DATA[1387,27] := 142.8095;
   DATA[1387,28] := 263.1056;
   DATA[1387,29] := 12.11228;
   DATA[1387,30] := 1.719687;
   DATA[1387,31] := 1.28705;
   DATA[1387,32] := 0.7355248;
   DATA[1387,33] := 0.3083624;
   DATA[1387,34] := 2.0;
   DATA[1387,35] := 249.5995;
   DATA[1387,36] := 1.601897;
   DATA[1387,37] := 188.4613;
   DATA[1387,38] := 0.000128152;
   DATA[1387,39] := 1.0;
   DATA[1388,1] := 813.5919;
   DATA[1388,2] := 1.0;
   DATA[1388,3] := 1.0;
   DATA[1388,4] := 262.5609;
   DATA[1388,5] := 8.46501;
   DATA[1388,6] := 318.1236;
   DATA[1388,8] := 1.0;
   DATA[1388,9] := 1.0;
   DATA[1388,10] := 1.0;
   DATA[1388,11] := 19.70357;
   DATA[1388,12] := 2.219902;
   DATA[1388,13] := 990.8116;
   DATA[1388,14] := 1.0;
   DATA[1388,15] := 2.0;
   DATA[1388,16] := 1.0;
   DATA[1388,17] := 1.0;
   DATA[1388,18] := 1.0;
   DATA[1388,19] := 2.0;
   DATA[1388,20] := 148.808;
   DATA[1388,21] := 153.4991;
   DATA[1388,22] := 1.709416;
   DATA[1388,23] := 779.9539;
   DATA[1388,24] := 2.0;
   DATA[1388,25] := 2.0;
   DATA[1388,26] := 7.87798;
   DATA[1388,27] := 142.8095;
   DATA[1388,28] := 263.1056;
   DATA[1388,29] := 12.11228;
   DATA[1388,30] := 1.718021;
   DATA[1388,31] := 1.280389;
   DATA[1388,32] := 0.7355248;
   DATA[1388,33] := 0.3083624;
   DATA[1388,34] := 2.0;
   DATA[1388,35] := 249.5995;
   DATA[1388,36] := 1.601897;
   DATA[1388,37] := 188.4613;
   DATA[1388,38] := 0.000128152;
   DATA[1388,39] := 1.0;
   DATA[1389,1] := 813.5527;
   DATA[1389,2] := 1.0;
   DATA[1389,3] := 1.0;
   DATA[1389,4] := 262.5609;
   DATA[1389,5] := 8.46501;
   DATA[1389,6] := 318.1236;
   DATA[1389,8] := 1.0;
   DATA[1389,9] := 1.0;
   DATA[1389,10] := 1.0;
   DATA[1389,11] := 19.76439;
   DATA[1389,12] := 2.219902;
   DATA[1389,13] := 990.0907;
   DATA[1389,14] := 1.0;
   DATA[1389,15] := 2.0;
   DATA[1389,16] := 1.0;
   DATA[1389,17] := 1.0;
   DATA[1389,18] := 1.0;
   DATA[1389,19] := 2.0;
   DATA[1389,20] := 148.808;
   DATA[1389,21] := 153.4991;
   DATA[1389,22] := 1.70916;
   DATA[1389,23] := 779.2617;
   DATA[1389,24] := 2.0;
   DATA[1389,25] := 2.0;
   DATA[1389,26] := 7.87798;
   DATA[1389,27] := 142.8095;
   DATA[1389,28] := 263.1056;
   DATA[1389,29] := 12.11228;
   DATA[1389,30] := 1.716483;
   DATA[1389,31] := 1.272192;
   DATA[1389,32] := 0.7355248;
   DATA[1389,33] := 0.3083624;
   DATA[1389,34] := 2.0;
   DATA[1389,35] := 249.5995;
   DATA[1389,36] := 1.601897;
   DATA[1389,37] := 188.4613;
   DATA[1389,38] := 0.000128152;
   DATA[1389,39] := 1.0;
   DATA[1390,1] := 813.5527;
   DATA[1390,2] := 1.0;
   DATA[1390,3] := 1.0;
   DATA[1390,4] := 262.5609;
   DATA[1390,5] := 8.46501;
   DATA[1390,6] := 318.1236;
   DATA[1390,8] := 1.0;
   DATA[1390,9] := 1.0;
   DATA[1390,10] := 1.0;
   DATA[1390,11] := 19.7836;
   DATA[1390,12] := 2.218493;
   DATA[1390,13] := 989.61;
   DATA[1390,14] := 1.0;
   DATA[1390,15] := 2.0;
   DATA[1390,16] := 1.0;
   DATA[1390,17] := 1.0;
   DATA[1390,18] := 1.0;
   DATA[1390,19] := 2.0;
   DATA[1390,20] := 148.808;
   DATA[1390,21] := 153.4991;
   DATA[1390,22] := 1.70916;
   DATA[1390,23] := 779.1464;
   DATA[1390,24] := 2.0;
   DATA[1390,25] := 2.0;
   DATA[1390,26] := 7.87798;
   DATA[1390,27] := 142.8095;
   DATA[1390,28] := 263.1056;
   DATA[1390,29] := 12.11228;
   DATA[1390,30] := 1.716483;
   DATA[1390,31] := 1.269502;
   DATA[1390,32] := 0.7355248;
   DATA[1390,33] := 0.3083624;
   DATA[1390,34] := 2.0;
   DATA[1390,35] := 249.5995;
   DATA[1390,36] := 1.601897;
   DATA[1390,37] := 188.4613;
   DATA[1390,38] := 0.000128152;
   DATA[1390,39] := 1.0;
   DATA[1391,1] := 813.1994;
   DATA[1391,2] := 1.0;
   DATA[1391,3] := 1.0;
   DATA[1391,4] := 262.5609;
   DATA[1391,5] := 8.46501;
   DATA[1391,6] := 318.1236;
   DATA[1391,8] := 1.0;
   DATA[1391,9] := 1.0;
   DATA[1391,10] := 1.0;
   DATA[1391,11] := 19.7836;
   DATA[1391,12] := 2.217468;
   DATA[1391,13] := 989.2896;
